// ---- DUTs/Communication/E_TaskName.TcDUT
{attribute 'qualified_only'}
{attribute 'strict'}
TYPE E_TaskName :
(
//(*
	//New
	EmptyTask :=0,
	ActivateRecipe							:=  1  	,
	ValidateRecipe                          :=  2   ,
	AlarmReset                              :=  3   ,
	ReadRFID                                :=  4   ,
	UpdateLCD                               :=  5   ,
	EnableModule                            :=  6   ,
	DisableModule                           :=  7   ,
	SetLogFileVerbosity                     :=  8   ,
	Initialize                              :=  9   ,
	Resume                                  :=  10  ,
	DoorOpen                                :=  11  ,
	DoorClose                               :=  12  ,
	DPSPower                                :=  13  ,
	UnitPresentCheck                        :=  14  ,
	TrayClamp                               :=  15  ,
	ChangeStackCount                        :=  16  ,
	BypassVision                            :=  17  ,
	TCCSessionRequest                       :=  18  ,
	TIUSlideOut                             :=  19  ,
	PrecisorSlideOut                        :=  20  ,
	SingulateTrayStacker                    :=  21  ,
	SingulateTrayStackerHalf                :=  22  ,
	SingulateTrayStackerRemaining           :=  23  ,
	StackUpTrayStacker                      :=  24  ,
	StopperUp                               :=  25  ,
	MoveConveyorForward                     :=  26  ,
	MoveConveyorBackward                    :=  27  ,
	MoveVisionShuttle                       :=  28  ,
	MoveUPortShuttle                        :=  29  ,
	UPortShuttleReady                       :=  30  ,
	MoveFlyoverShuttle                      :=  31  ,
	FlyoverShuttlePick                      :=  32  ,
	FlyoverShuttlePlace                     :=  33  ,
	MoveTrayScanShuttle                     :=  34  ,
	MoveTrayScanShuttleLifter               :=  35  ,
	EportLatch                              :=  36  ,
	GantryPickAndPlace                      :=  37  ,
	TBOTPickAndPlace                        :=  38  ,
	AutoTeach                               :=  39  ,
	Jog                                     :=  40  ,
	ApplyTeachData                          :=  41  ,
	AbortTeach                              :=  42  ,
	WriteRFIDData                           :=  43  ,
	MoveGantry                              :=  44  ,
	MoveTBOT                                :=  45  ,
	MoveTBOTRetry                           :=  46  ,
	MoveTBOTCancel                          :=  47  ,
	TBOTPickAndPlaceRetry                   :=  48  ,
	TBOTPickAndPlaceCancel                  :=  49  ,
	MoveGantryRetry                         :=  50  ,
	MoveGantryCancel                        :=  51  ,
	GantryPickAndPlaceRetry                 :=  52  ,
	GantryPickAndPlaceCancel                :=  53  ,
	SingulateTrayStackerRetry               :=  54  ,
	SingulateTrayStackerCancel              :=  55  ,
	SingulateTrayStackerHalfRetry           :=  56  ,
	SingulateTrayStackerHalfCancel          :=  57  ,
	SingulateTrayStackerRemainingRetry      :=  58  ,
	SingulateTrayStackerRemainingCancel     :=  59  ,
	StackUpTrayStackerRetry                 :=  60  ,
	StackUpTrayStackerCancel                :=  61  ,
	MoveConveyorForwardRetry                :=  62  ,
	MoveConveyorForwardCancel               :=  63  ,
	MoveConveyorBackwardRetry               :=  64  ,
	MoveConveyorBackwardCancel              :=  65  ,
	MoveVisionShuttleRetry                  :=  66  ,
	MoveVisionShuttleCancel                 :=  67  ,
	MoveUPortShuttleRetry                   :=  68  ,
	MoveUPortShuttleCancel                  :=  69  ,
	MoveFlyoverShuttleRetry                 :=  70  ,
	MoveFlyoverShuttleCancel                :=  71  ,
	MoveTrayScanShuttleRetry                :=  72  ,
	MoveTrayScanShuttleCancel               :=  73  ,
	MoveTrayScanShuttleLifterRetry          :=  74  ,
	MoveTrayScanShuttleLifterCancel         :=  75  ,
	Cancel                                  :=  76  ,
	TIUSlideOutRetry                        :=  77  ,
	TIUSlideOutCancel                       :=  78  ,
	MoveTTSShuttle                          :=  79  ,
	MoveTTSShuttleRetry                     :=  80  ,
	MoveTTSShuttleCancel                    :=  81  ,
	SingulateTrayLatchRemaining             :=  82  ,
	SingulateTrayLatchRemainingRetry        :=  83  ,
	SingulateTrayLatchRemainingCancel       :=  84  ,
	SingulateTrayLatch                      :=  85  ,
	SingulateTrayLatchRetry                 :=  86  ,
	SingulateTrayLatchCancel                :=  87  ,
	StackUpTrayLatch                        :=  88  ,
	StackUpTrayLatchRetry                   :=  89  ,
	StackUpTrayLatchCancel                  :=  90  ,
	SingulateCylinderTray                   :=  91  ,
	SingulateCylinderTrayRetry              :=  92  ,
	SingulateCylinderTrayCancel             :=  93  ,
	StackUpCylinderTray                     :=  94  ,
	StackUpCylinderTrayRetry                :=  95  ,
	StackUpCylinderTrayCancel               :=  96  ,
	SetUPortBlinkRate                       :=  97  ,
	TBotUnitPresentCheck                    :=  98  ,
	AP240ACPOWER                            :=  99  ,
	TesterAirValve                          :=  100 ,
	APAirValve                              :=  101 ,
	DrawerUp                                :=  102 ,
	SetBlinkRate							:=  103 ,
	TIUSocketCoolingAir						:=  104	,
	StackDownTrayStacker					:=	105	,
	StackDownTrayStackerRetry				:=	106	,
	StackDownTrayStackerCancel				:=	107	,
	StackDownTrayStackerRemaining			:=	108	,
	StackDownTrayStackerRemainingRetry		:=	109	,
	StackDownTrayStackerRemainingCancel		:=	110	,
	TTSShuttlePickPlace						:=	111	,
	TTSShuttlePickPlaceCancel				:=	112	,
	TTSShuttlePickPlaceRetry				:=	113	,
	HstTbotPickAndPlace						:=	114	,
	HstTbotPickAndPlaceRetry				:=	115	,
	HstTbotPickAndPlaceCancel				:=	116	,
	StackDownTrayStackerHalf				:=	117	,
	StackDownTrayStackerHalfRetry			:=	118	,
	StackDownTrayStackerHalfCancel			:=	119	,
	SetStackerBlinkRate						:=	120	,
	Ap48DCPower								:=	121	,
	BPAirValve								:=	122	,
	APPCWValve								:=	123	,
	CellLTIMValve							:=	124	,
	MainPCWValve							:=	125	,
	MainOFAValve							:=	126	,
	CmdPower								:=	127	,
	SetSolenoidValves						:=	128	,
	Secondary24VPower						:=	131

);
END_TYPE

// ---- DUTs/Communication/ST_Command.TcDUT
TYPE ST_Command :
STRUCT
	sLogName	: STRING(81);
	eTaskName	: E_TaskName;
	eModuleID	: E_ModuleID;
	iParam		: ARRAY [1..NO_OF_INT_PARAM] OF DINT;
	sParam		: ARRAY [1..NO_OF_STRING_PARAM] OF STRING;
	bParam		: ARRAY [1..NO_OF_BOOL_PARAM] OF BOOL;
	dParam		: ARRAY [1..NO_OF_LREAL_PARAM] OF LREAL;
END_STRUCT
END_TYPE

// ---- DUTs/Communication/ST_Event.TcDUT
TYPE ST_Event :
STRUCT
	sLogName	: STRING(81);
	eEventName	: E_EventName;
	eModuleID	: E_ModuleID;
	iParam		: ARRAY [1..NO_OF_INT_PARAM] OF DINT;
	sParam		: ARRAY [1..NO_OF_STRING_PARAM] OF STRING;
	bParam		: ARRAY [1..NO_OF_BOOL_PARAM] OF BOOL; 
	dParam		: ARRAY [1..NO_OF_LREAL_PARAM] OF LREAL; 
	sFailReason	: STRING(81);
END_STRUCT
END_TYPE

// ---- DUTs/Communication/ST_EventQueue.TcDUT
TYPE ST_EventQueue :
STRUCT
	Queue: ARRAY [1..255] OF ST_Event;	//255 queue buffers
	Count: UINT := 0;
END_STRUCT
END_TYPE

// ---- DUTs/Communication/ST_TACommands.TcDUT
TYPE ST_TACommands :
STRUCT
	arrTACommands : ARRAY  [1..NO_OF_CMD_BUFFER] OF ST_Command;
		
END_STRUCT
END_TYPE

// ---- DUTs/Communication/ST_TAEvents.TcDUT
TYPE ST_TAEvents :
STRUCT
	arrTAEvents : ARRAY [1..NO_OF_EVENT_BUFFER]  OF ST_Event;
	
END_STRUCT
END_TYPE

// ---- DUTs/Enum/E_BackdoorState_1.TcDUT
TYPE E_BackdoorState_1 :
(
	eDisable := 0,
	eForce_On :=1,
	eForce_Off := 2
);
END_TYPE

// ---- DUTs/Enum/E_ModuleID_1.TcDUT
TYPE E_ModuleID_1 :
(
	eNull := 0,

//Uport
	eUport1,
	eUport2,
	eUport1Stk,
	eUport2Stk,

//Uport shuttle
	eUShuttle1,
	eUShuttle2,
	eUShuttle1Cny,
	eUShuttle2Cny,
	eUShuttle1Prk,
	eUShuttle2Prk,

//LP Lane	
	eLP1,
	eLP2,
	eLP3,
	eLP4,
	eLP5,
	eLP6,
	eLP7,
	eLP8,
	
	eLP1Stk1,
	eLP2Stk1,
	eLP3Stk1,
	eLP4Stk1,
	eLP5Stk1,
	eLP6Stk1,
	eLP7Stk1,
	eLP8Stk1,

	eLP1Stk2,
	eLP2Stk2,
	eLP3Stk2,
	eLP4Stk2,
	eLP5Stk2,
	eLP6Stk2,
	eLP7Stk2,
	eLP8Stk2,
	
		eLP1Stk1Lift,
		eLP2Stk1Lift,
		eLP3Stk1Lift,
		eLP4Stk1Lift,
		eLP5Stk1Lift,
		eLP6Stk1Lift,
		eLP7Stk1Lift,
		eLP8Stk1Lift,
	
		eLP1Stk2Lift,
		eLP2Stk2Lift,
		eLP3Stk2Lift,
		eLP4Stk2Lift,
		eLP5Stk2Lift,
		eLP6Stk2Lift,
		eLP7Stk2Lift,
		eLP8Stk2Lift,

		eLP1Stk1Cny,
		eLP2Stk1Cny,
		eLP3Stk1Cny,
		eLP4Stk1Cny,
		eLP5Stk1Cny,
		eLP6Stk1Cny,
		eLP7Stk1Cny,
		eLP8Stk1Cny,
	
		eLP1Stk2Cny,
		eLP2Stk2Cny,
		eLP3Stk2Cny,
		eLP4Stk2Cny,
		eLP5Stk2Cny,
		eLP6Stk2Cny,
		eLP7Stk2Cny,
		eLP8Stk2Cny,

	eLP1Eport,
	eLP2Eport,
	eLP3Eport,
	eLP4Eport,
	eLP5Eport,
	eLP6Eport,
	eLP7Eport,
	eLP8Eport,	

		eLP1EportStk,
		eLP2EportStk,
		eLP3EportStk,
		eLP4EportStk,
		eLP5EportStk,
		eLP6EportStk,
		eLP7EportStk,
		eLP8EportStk,
	
		eLP1EportCny,
		eLP2EportCny,
		eLP3EportCny,
		eLP4EportCny,
		eLP5EportCny,
		eLP6EportCny,
		eLP7EportCny,
		eLP8EportCny,
		
		eLP1EportGrip,
		eLP2EportGrip,
		eLP3EportGrip,
		eLP4EportGrip,
		eLP5EportGrip,
		eLP6EportGrip,
		eLP7EportGrip,
		eLP8EportGrip,		
		
	eLP1Shuttle,
	eLP2Shuttle,
	eLP3Shuttle,
	eLP4Shuttle,
	eLP5Shuttle,
	eLP6Shuttle,
	eLP7Shuttle,
	eLP8Shuttle,

//TTS
	eTTS1,
	eTTS2,

	eTTS1Prk,
	eTTS2Prk,

//Vision
	eVision1,
	eVision2,
	
	eVision1Prk,
	eVision2Prk,
	
//**********************
	eUport,
	eUportStk,
	
	eUShuttle,
	eUShuttleCny,
	eUShuttlePrk,

	eLP,
	eLPStk,
	eLPStk1,
	eLPStk2,
	eLPStkCny,
	eLPStkLift,
	eLPEport,
	
	eTTS,
	eTTSPrk,
	
	eVision,
	eVisionPrk,
	
	eLPEportLatch,
	eLPEportTTS,
	
	ePNBLatch,
	ePNBSby,
	ePNB
	
	
);
END_TYPE

// ---- DUTs/Enum/E_ProcessState.TcDUT
TYPE E_ProcessState :
(
	eUNKNOWN:=0,
	eINIT,		//During Init
	//eIDLE,
	//eIDLEAL,
	//eSETGUP,
	//eREADY,
	eAWAITGCMD,	//After Done = Idle
	eLOADG,		//Processing
    //eALARM,
	ePAUSE,		//Aft Alm Rst
	//eTARESUME,
	eALPAUSED//,	//During Alm
	//eCHECKG,
	//eCOMPLETE
	
	
);
END_TYPE

// ---- DUTs/Enum/E_ProcessStep.TcDUT
TYPE E_ProcessStep :
(
	eSeqReset:=1,
	eDataInput,
	eExecuting,
	eSeqCompleted,
	eSeqError,
	eSeqCancel	
);
END_TYPE

// ---- DUTs/Enum/E_SeqSts_1.TcDUT
TYPE E_SeqSts_1 :
(
	eNull := -1,
	eInit := 0,
	ePreSanityCheck,
	eSanityCheck,
	eSanityCheck2,
	eTrayCount,

	//hw trigger
	eMotorZVelMove,	//Velosity move
	eMotorZVelMoveTeach,
	eMotorXVelMove,
	eMotorYVelMove,
	eMotorZHalt,
	eMotorXHalt,
	eMotorYHalt,
	eMotorCnyMove,
	eMotorCnyMoveSlow,
	eMotorCnyHalt,
	
// ^^^^Skip seq step till eMotorCnyHalt^^^^

	eMotorZAbsMove,	//Absolute move
	eMotorXAbsMove,
	eMotorYAbsMove,
	eMotorZRelMove,	//Relative move
	eMotorXRelMove,
	eMotorYRelMove,
	eClamp,
	eUnclamp,
	eLatch,
	eUnlatch,
	eEportLatch,
	eEportUnlatch,
	eStopperUp,
	eStopperDwn,
	eShutterOpen,
	eShutterClose,
	
	eMotorXReset,
	eMotorYReset,
	eMotorZReset,
	
	eMotorXPowerOn,
	eMotorYPowerOn,
	eMotorZPowerOn,
	
	eMotorXHome,
	eMotorYHome,
	eMotorZHome,
	
	eMotorConyReset,
	eMotorConyPowerOn,
	eMotorConyHome,
	
	eMotorZAbsMoveSbyPos,
	eMotorZAbsMoveLatchPos,
	eMotorZAbsMoveLiftPos,
	eMotorZAbsMoveTopPos,
	eMotorZAbsMoveCountSensorPos,
	eMotorZAbsMoveEportTopPos,
	eAutoTeachCalc,
		
	
	
	eCylJackUp,
	eCylJackDown,
	
	eHomeStacker,
	eHomeConveyer,
	eHomeUport,
	
	eReset,
	eExecute,
	eAlarmed,
	
	eDone :=100
	
);
END_TYPE

// ---- DUTs/E_BackdoorState.TcDUT
TYPE E_BackdoorState :
(
	eDisable := 0,
	eForce_On :=1,
	eForce_Off := 2
);
END_TYPE

// ---- DUTs/HMI/ST_BypassTII.TcDUT
TYPE ST_BypassTII :
STRUCT
	bHMITIIByPassArray:ARRAY[1..NO_OF_TII_SENSOR] OF BOOL;
END_STRUCT
END_TYPE

// ---- DUTs/ModuleState/EnableDisable/E_State.TcDUT
TYPE E_State :
(
	// Disabled
	eDisabled :=0,
	// Enabled
	eEnabled
);
END_TYPE

// ---- DUTs/ModuleState/EnableDisable/ST_LPState.TcDUT
TYPE ST_LPState :
STRUCT
	// LoadPort module state 
	//arrLPSubModule : ARRAY [1..(.NO_OF_LANES)] OF ST_TCSubModuleState;
	
	
//	EmptyStacker : ARRAY [1..(.NO_OF_STACKERS_IN_EMPTYSTK)] OF E_State := [(.NO_OF_STACKERS_IN_EMPTYSTK)(E_State.eEnabled)];
	// Vision Shuttle 
	//VisionShuttle : E_State := E_State.eEnabled;
END_STRUCT
END_TYPE

// ---- DUTs/ModuleState/EnableDisable/ST_LPTTS_State.TcDUT
TYPE ST_LPTTS_State :
STRUCT
	// LoadPort module state , 2 LPs
	arrLoadPort: ARRAY [1..(.NO_OF_LPS)] OF ST_LPState;
	// TTS moduel state
	stTTS: ST_TTS_State;
		
END_STRUCT
END_TYPE

// ---- DUTs/ModuleState/EnableDisable/ST_TCSubModuleState.TcDUT
TYPE ST_TCSubModuleState :
STRUCT
	Tester							: E_State := E_State.eEnabled;
	TCSite							: ARRAY [1..(.NO_OF_TC_SITE)] OF ST_TCSiteState;
END_STRUCT
END_TYPE

// ---- DUTs/ModuleState/EnableDisable/ST_TCSiteState.TcDUT
TYPE ST_TCSiteState :
STRUCT
	TCU						: E_State	:= E_State.eEnabled;
	TIERII					: E_State	:= E_State.eEnabled;
END_STRUCT
END_TYPE

// ---- DUTs/ModuleState/EnableDisable/ST_TTS_State.TcDUT
TYPE ST_TTS_State :
STRUCT
	// TTS moduel state
	arrTTSLane: ARRAY [1..3] OF E_State := [(3)(E_State.eEnabled)];
END_STRUCT
END_TYPE

// ---- DUTs/ModuleState/EPT/E_EPT.TcDUT
TYPE E_EPT :
(
	// Unknown, Alarm, Paused, Aborting, Claibration, Manual
	eBlocked :=0,
	// Idle
	eIdle,
	// Initialize, SettingUp, Ready, Executing, Checking
	eBusy 
);
END_TYPE

// ---- DUTs/ModuleState/EPT/ST_LPTTS_EPT.TcDUT
TYPE ST_LPTTS_EPT :
STRUCT
	// LoadPort module state , 2 LPs
	//arrLoadPort: ARRAY [1..(.NO_OF_LPS)] OF ST_LP_EPT;
	// TTS moduel state
	stTTS: ST_TTS_EPT;
		
END_STRUCT
END_TYPE

// ---- DUTs/ModuleState/EPT/ST_TCUEPT.TcDUT
TYPE ST_TCUEPT :
STRUCT
	// LoadPort module state 
	//arrLPSubModule : ARRAY [1..(.NO_OF_LANES)] OF ST_LP_SubModuleEPT;
	// Vision Shuttle 
	TCU : E_EPT;
END_STRUCT
END_TYPE

// ---- DUTs/ModuleState/EPT/ST_TCSubModuleEPT.TcDUT
TYPE ST_TCSubModuleEPT :
STRUCT
	TCSite: ARRAY [1..(.NO_OF_TC_SITE)] OF ST_TCUEPT;
END_STRUCT
END_TYPE

// ---- DUTs/ModuleState/EPT/ST_TC_EPT.TcDUT
TYPE ST_TC_EPT :
STRUCT
	eTCEpt:E_EPT;
	
END_STRUCT
END_TYPE

// ---- DUTs/ModuleState/EPT/ST_TTS_EPT.TcDUT
TYPE ST_TTS_EPT :
STRUCT
	// TTS State
	eTTS: E_EPT;
	// TTS moduel state
	arrTTSLane: ARRAY [1..3] OF E_EPT;
END_STRUCT
END_TYPE

// ---- DUTs/ST_StepMode.TcDUT
TYPE ST_StepMode :
STRUCT
	bStepMode: BOOL;  //module in step mode
	bStep	 : BOOL;  //Step by step
END_STRUCT
END_TYPE

// ---- DUTs/ST_DebugStation.TcDUT
TYPE ST_DebugStation :
STRUCT
		stGblDBStnParam		: ST_DebugStationSeqParam;
		fbDBStnSeq			: FB_DebugStationSeq;
END_STRUCT
END_TYPE

// ---- DUTs/ST_TCMultilevel.TcDUT
TYPE ST_TCMultilevel :
STRUCT
	
		stGblParam							: ST_TCMultiLevelSeqParam;
		fbTCMultiLevelSeq					: FB_TCMultiLevelSeq;
		
END_STRUCT
END_TYPE

// ---- DUTs/ST_TCShuttlePOC.TcDUT
TYPE ST_TCShuttlePOC :
STRUCT
	
		stGblParam: ST_TCSeqParam;
		fbTCShuttlePOCSeq: FB_TCShuttlePOCSeq;

END_STRUCT
END_TYPE

// ---- DUTs/ST_TCLevel.TcDUT
TYPE ST_TCLevel :
STRUCT
	
		stGblParam: ST_TCSeqParam;
		fbTCLevelSeq: FB_TCLevelSeq;
		
END_STRUCT
END_TYPE

// ---- GVLs/GVL_CONSTANTS.TcGVL
VAR_GLOBAL CONSTANT

	// This function has been automatically generated from the project information.
	stLibVersion_TC : ST_LibVersion := (iMajor := 0, iMinor := 0, iBuild := 0, iRevision := 0, sVersion := '2.0.5');

	LA_LEVEL_MODULE_ID : ARRAY [1..NO_OF_LEVEL] OF E_ModuleID  := [	E_ModuleID.CELL_LA101_TESTER, E_ModuleID.CELL_LA201_TESTER, E_ModuleID.CELL_LA301_TESTER,
																	E_ModuleID.CELL_LA401_TESTER, E_ModuleID.CELL_LA501_TESTER, E_ModuleID.CELL_LA601_TESTER];
	LB_LEVEL_MODULE_ID : ARRAY [1..NO_OF_LEVEL] OF E_ModuleID  := [	E_ModuleID.CELL_LB101_TESTER, E_ModuleID.CELL_LB201_TESTER, E_ModuleID.CELL_LB301_TESTER,
																	E_ModuleID.CELL_LB401_TESTER, E_ModuleID.CELL_LB501_TESTER, E_ModuleID.CELL_LB601_TESTER];
	LC_LEVEL_MODULE_ID : ARRAY [1..NO_OF_LEVEL] OF E_ModuleID  := [	E_ModuleID.CELL_LC101_TESTER, E_ModuleID.CELL_LC201_TESTER, E_ModuleID.CELL_LC301_TESTER,
																	E_ModuleID.CELL_LC401_TESTER, E_ModuleID.CELL_LC501_TESTER, E_ModuleID.CELL_LC601_TESTER];
	RA_LEVEL_MODULE_ID : ARRAY [1..NO_OF_LEVEL] OF E_ModuleID  := [	E_ModuleID.CELL_RA101_TESTER, E_ModuleID.CELL_RA201_TESTER, E_ModuleID.CELL_RA301_TESTER,
																	E_ModuleID.CELL_RA401_TESTER, E_ModuleID.CELL_RA501_TESTER, E_ModuleID.CELL_RA601_TESTER];
	RB_LEVEL_MODULE_ID : ARRAY [1..NO_OF_LEVEL] OF E_ModuleID  := [	E_ModuleID.CELL_RB101_TESTER, E_ModuleID.CELL_RB201_TESTER, E_ModuleID.CELL_RB301_TESTER,
																	E_ModuleID.CELL_RB401_TESTER, E_ModuleID.CELL_RB501_TESTER, E_ModuleID.CELL_RB601_TESTER];
	RC_LEVEL_MODULE_ID : ARRAY [1..NO_OF_LEVEL] OF E_ModuleID  := [	E_ModuleID.CELL_RC101_TESTER, E_ModuleID.CELL_RC201_TESTER, E_ModuleID.CELL_RC301_TESTER,
																	E_ModuleID.CELL_RC401_TESTER, E_ModuleID.CELL_RC501_TESTER, E_ModuleID.CELL_RC601_TESTER];	
														
	LA_FRONT_DOOR_MODULE_ID : ARRAY [1..2] OF E_ModuleID  := [E_ModuleID.CELL_LA101_TESTER_FRONT, E_ModuleID.CELL_LA201_TESTER_FRONT];	
	
//<ForEnDisMod>
	ARR_LA_TST_MODULE_ID : ARRAY [1..6] OF E_ModuleID  := [E_ModuleID.CELL_LA101_TESTER, E_ModuleID.CELL_LA201_TESTER, E_ModuleID.CELL_LA201_TESTER, 
														   E_ModuleID.CELL_LA401_TESTER, E_ModuleID.CELL_LA501_TESTER, E_ModuleID.CELL_LA601_TESTER];	
	ARR_LB_TST_MODULE_ID : ARRAY [1..6] OF E_ModuleID  := [E_ModuleID.CELL_LB101_TESTER, E_ModuleID.CELL_LB201_TESTER, E_ModuleID.CELL_LB201_TESTER, 
														   E_ModuleID.CELL_LB401_TESTER, E_ModuleID.CELL_LB501_TESTER, E_ModuleID.CELL_LB601_TESTER];	
	ARR_LC_TST_MODULE_ID : ARRAY [1..6] OF E_ModuleID  := [E_ModuleID.CELL_LC101_TESTER, E_ModuleID.CELL_LC201_TESTER, E_ModuleID.CELL_LC201_TESTER, 
														   E_ModuleID.CELL_LC401_TESTER, E_ModuleID.CELL_LC501_TESTER, E_ModuleID.CELL_LC601_TESTER];															   
	ARR_RA_TST_MODULE_ID : ARRAY [1..6] OF E_ModuleID  := [E_ModuleID.CELL_RA101_TESTER, E_ModuleID.CELL_RA201_TESTER, E_ModuleID.CELL_RA201_TESTER, 
													   	   E_ModuleID.CELL_RA401_TESTER, E_ModuleID.CELL_RA501_TESTER, E_ModuleID.CELL_RA601_TESTER];	
	ARR_RB_TST_MODULE_ID : ARRAY [1..6] OF E_ModuleID  := [E_ModuleID.CELL_RB101_TESTER, E_ModuleID.CELL_RB201_TESTER, E_ModuleID.CELL_RB201_TESTER, 
													       E_ModuleID.CELL_RB401_TESTER, E_ModuleID.CELL_RB501_TESTER, E_ModuleID.CELL_RB601_TESTER];	
	ARR_RC_TST_MODULE_ID : ARRAY [1..6] OF E_ModuleID  := [E_ModuleID.CELL_RC101_TESTER, E_ModuleID.CELL_RC201_TESTER, E_ModuleID.CELL_RC201_TESTER, 
														   E_ModuleID.CELL_RC401_TESTER, E_ModuleID.CELL_RC501_TESTER, E_ModuleID.CELL_RC601_TESTER];		
														   
	ARR_LA_TCU_MODULE_ID : ARRAY [1..6] OF E_ModuleID  := [E_ModuleID.CELL_LA101_AP, E_ModuleID.CELL_LA201_AP, E_ModuleID.CELL_LA201_AP, 
														   E_ModuleID.CELL_LA401_AP, E_ModuleID.CELL_LA501_AP, E_ModuleID.CELL_LA601_AP];	
	ARR_LB_TCU_MODULE_ID : ARRAY [1..6] OF E_ModuleID  := [E_ModuleID.CELL_LB101_AP, E_ModuleID.CELL_LB201_AP, E_ModuleID.CELL_LB201_AP, 
														   E_ModuleID.CELL_LB401_AP, E_ModuleID.CELL_LB501_AP, E_ModuleID.CELL_LB601_AP];	
	ARR_LC_TCU_MODULE_ID : ARRAY [1..6] OF E_ModuleID  := [E_ModuleID.CELL_LC101_AP, E_ModuleID.CELL_LC201_AP, E_ModuleID.CELL_LC201_AP, 
														   E_ModuleID.CELL_LC401_AP, E_ModuleID.CELL_LC501_AP, E_ModuleID.CELL_LC601_AP];															   
	ARR_RA_TCU_MODULE_ID : ARRAY [1..6] OF E_ModuleID  := [E_ModuleID.CELL_RA101_AP, E_ModuleID.CELL_RA201_AP, E_ModuleID.CELL_RA201_AP, 
													   	   E_ModuleID.CELL_RA401_AP, E_ModuleID.CELL_RA501_AP, E_ModuleID.CELL_RA601_AP];	
	ARR_RB_TCU_MODULE_ID : ARRAY [1..6] OF E_ModuleID  := [E_ModuleID.CELL_RB101_AP, E_ModuleID.CELL_RB201_AP, E_ModuleID.CELL_RB201_AP, 
													       E_ModuleID.CELL_RB401_AP, E_ModuleID.CELL_RB501_AP, E_ModuleID.CELL_RB601_AP];	
	ARR_RC_TCU_MODULE_ID : ARRAY [1..6] OF E_ModuleID  := [E_ModuleID.CELL_RC101_AP, E_ModuleID.CELL_RC201_AP, E_ModuleID.CELL_RC201_AP, 
														   E_ModuleID.CELL_RC401_AP, E_ModuleID.CELL_RC501_AP, E_ModuleID.CELL_RC601_AP];		


	ARR_LA_TII_MODULE_ID : ARRAY [1..6] OF E_ModuleID  := [E_ModuleID.CELL_LA101_TIERII, E_ModuleID.CELL_LA201_TIERII, E_ModuleID.CELL_LA201_TIERII, 
														   E_ModuleID.CELL_LA401_TIERII, E_ModuleID.CELL_LA501_TIERII, E_ModuleID.CELL_LA601_TIERII];	
	ARR_LB_TII_MODULE_ID : ARRAY [1..6] OF E_ModuleID  := [E_ModuleID.CELL_LB101_TIERII, E_ModuleID.CELL_LB201_TIERII, E_ModuleID.CELL_LB201_TIERII, 
														   E_ModuleID.CELL_LB401_TIERII, E_ModuleID.CELL_LB501_TIERII, E_ModuleID.CELL_LB601_TIERII];	
	ARR_LC_TII_MODULE_ID : ARRAY [1..6] OF E_ModuleID  := [E_ModuleID.CELL_LC101_TIERII, E_ModuleID.CELL_LC201_TIERII, E_ModuleID.CELL_LC201_TIERII, 
														   E_ModuleID.CELL_LC401_TIERII, E_ModuleID.CELL_LC501_TIERII, E_ModuleID.CELL_LC601_TIERII];															   
	ARR_RA_TII_MODULE_ID : ARRAY [1..6] OF E_ModuleID  := [E_ModuleID.CELL_RA101_TIERII, E_ModuleID.CELL_RA201_TIERII, E_ModuleID.CELL_RA201_TIERII, 
													   	   E_ModuleID.CELL_RA401_TIERII, E_ModuleID.CELL_RA501_TIERII, E_ModuleID.CELL_RA601_TIERII];	
	ARR_RB_TII_MODULE_ID : ARRAY [1..6] OF E_ModuleID  := [E_ModuleID.CELL_RB101_TIERII, E_ModuleID.CELL_RB201_TIERII, E_ModuleID.CELL_RB201_TIERII, 
													       E_ModuleID.CELL_RB401_TIERII, E_ModuleID.CELL_RB501_TIERII, E_ModuleID.CELL_RB601_TIERII];	
	ARR_RC_TII_MODULE_ID : ARRAY [1..6] OF E_ModuleID  := [E_ModuleID.CELL_RC101_TIERII, E_ModuleID.CELL_RC201_TIERII, E_ModuleID.CELL_RC201_TIERII, 
														   E_ModuleID.CELL_RC401_TIERII, E_ModuleID.CELL_RC501_TIERII, E_ModuleID.CELL_RC601_TIERII];		
														   
//</ForEnDisMod>														  


													
	ARR_AMS_NET_ID : ARRAY [1..NO_OF_COLUMN] OF STRING := [	'192.168.1.4.1.1',
															'192.168.1.5.1.1', 
															'192.168.1.6.1.1',
															'192.168.1.14.1.1',
															'192.168.1.15.1.1', 
															'192.168.1.16.1.1'];	
		
	ARR_COL_MOD_ID : ARRAY [1..NO_OF_COLUMN] OF E_ModuleID := [	E_ModuleID.COLUMN_LA,
																E_ModuleID.COLUMN_LB,
																E_ModuleID.COLUMN_LC,
																E_ModuleID.COLUMN_RA,
																E_ModuleID.COLUMN_RB,
																E_ModuleID.COLUMN_RC];										
	TIIAlmText : ARRAY[1..NO_OF_TII_SENSOR] OF STRING :=
	[
	 	'AP_Not_Present'					,	
	 	'APPower_Not_On'	    			,
	 	'AP_Not_Ready' 		    			,
	 	'APDeactuatedPLC_Not_On' 			,
	 	'APDeactuatedHwr_Not_On' 			,
	 	'CellFluid_Leakage1' 				,
	 	'CellFluid_Leakage2' 				,
	 	'Cell_GroundFault' 					,
	 	'Tester_Not_Present' 				,
	 	'TesterPower_Not_On' 				,
	 	'Tester_not_ready'					,
	 	'TCCellDoor_Not_Locked'				,
	 	'TesterLatches_Not_Closed' 			,
	 	'TBOT_TC_ACPower_Off_Signal' 		,
		'DS_Facility_EAP_ACPower_Signal'	,
		'FrontDoorLockSignalNotDetected'	,
	 	'TCDrawerCylExtendRS_Not_On' 		,
	 	'TCDrawerCylRetractRS_Not_On'		,
		'TCDrawerUpSignal_not_on'			,
		'TCDrawerDownSignal_not_on'		    	
	];
	
	EAPAlmText : ARRAY[1..NO_OF_LEVEL,1..NO_OF_EAP_ALARM] OF STRING :=
	[
	 	'TBOT EAP ALARM_1'				,	
	 	'TBOT EAP ALARM_2'				,
	 	'TBOT EAP ALARM_3'				,
	 	'TBOT EAP ALARM_4'				,
	 	'TBOT EAP ALARM_5'				,
	 	'TBOT EAP ALARM_6'				,
	 	'TBOT EAP ALARM_7'				,
	 	'TBOT EAP ALARM_8'				,
	 	'TBOT EAP ALARM_9'				,
	 	'TBOT EAP ALARM_10'			
	];
	 
	SysAlmText : ARRAY[1..NO_OF_COMMON_SENSOR] OF STRING :=
	[
	 	'Column_PCWLeakage',
	 	'AllTCDrawer_Not_In_Cell',       
	 	'ipTbotDoorClosedSignal'
	];
	
	DBStnSysAlmText : ARRAY[1..NO_OF_DBCOL_ALARM] OF STRING :=
	[
	 	'SystemPCWLeakageAlarm',
	 	'SystemPCWSupplyLeakageAlarm',       
	 	'SystemPCWReturnLeakageAlarm',
	 	'CriticalCondensationAlarm',
	 	'6BarLowOFAAirPressureAlarm'
	];
															
	NO_OF_COMMON_SENSOR 						: UINT	:= 3;
	NO_OF_TII_SENSOR 							: UINT	:= 30;
	NO_OF_ALARM_TAG								: UINT 	:= 50;
	NO_OF_DC_CELL_LEVEL							: UINT	:= 2;
	NO_OF_LEVEL 								: UINT 	:= 6;
	NO_OF_COLUMN 								: UINT 	:= 6;
	NO_OF_TC_SITE								: UINT	:= 1;
	NO_OF_SENSORS 								: UINT 	:= 20;
	NO_OF_BTNLED								: INT	:= 5;
	NO_OF_EAP_ALARM								: INT	:= 10;
	NO_OF_DBCOL_ALARM							: INT	:= 10;
	
	//Path Setting
	LOGFILEPATHTC1 :STRING(30) := 'D:/ControllerLog/Level1/';
	LOGFILEPATHTC2 :STRING(30) := 'D:/ControllerLog/Level2/';
	LOGFILEPATHTC3 :STRING(30) := 'D:/ControllerLog/Level3/';
	LOGFILEPATHTC4 :STRING(30) := 'D:/ControllerLog/Level4/';
	LOGFILEPATHTC5 :STRING(30) := 'D:/ControllerLog/Level5/';
	
	//Log verbosity
	LOG_LEVEL_ERROR   : INT := 5;
	LOG_LEVEL_WARNING : INT := 4;
	LOG_LEVEL_MESSAGE : INT := 3;
	LOG_LEVEL_INFO    : INT := 2;
	LOG_LEVEL_DEBUG   : INT := 1;
	
	NO_OF_CMD_BUFFER : INT := 30;
	NO_OF_EVENT_BUFFER : INT := 30;
		
	NO_OF_INT_PARAM : INT := 10;
	NO_OF_STRING_PARAM :INT := 5;
	NO_OF_BOOL_PARAM :INT := 32;
	NO_OF_LREAL_PARAM :INT := 10;


	MODULEID_ERROR : STRING := 'Module ID not correct';

	NO_OF_LIB_ALARM:INT:=30;
	NO_OF_TA_ALARM: INT:=100;
	NO_OF_ALARM_PER_LEVEL : INT := 100;
END_VAR
VAR_GLOBAL
	lrTest: REAL;
END_VAR

// ---- GVLs/GVL_EAP.TcGVL
//{attribute 'qualified_only'}
VAR_GLOBAL
	stEAP:ST_EAP;
	stDCEAP:ST_DCEAP;
	DS_Facility_eapShutOffAllACPower					AT %I* :BOOL; // shut off Tester and AP AC Power, 0: On, 1: Off //only for debug cart and station
END_VAR

// ---- GVLs/GVL_Motor.TcGVL
//{attribute 'qualified_only'}
VAR_GLOBAL
	GVL_DUT_TC_AP240ACPower					: DUT_Cylinder;
	GVL_DUT_DC_AP240ACPower					: DUT_Cylinder;
END_VAR

// ---- GVLs/GVL_Process.TcGVL
//{attribute 'qualified_only'}
VAR_GLOBAL
	Sec_P						: BOOL;
	DewPoint_Warning			: BOOL;
	DewPoint_Alarm				: BOOL;
	DewPoint_Abort				: BOOL;
	OFA6Bar_Warning				: BOOL;
	OFA6Bar_Alarm				: BOOL;
	OFA6Bar_Abort				: BOOL;
	
	DewPoint_Warning_Timer		: UDINT	:= 300;
	DewPoint_Alarm_Timer		: UDINT	:= 60;
	DewPoint_Abort_Timer		: UDINT	:= 60;
	OFA6Bar_Warning_Timer		: UDINT	:= 300;
	OFA6Bar_Alarm_Timer			: UDINT	:= 60;
	OFA6Bar_Abort_Timer			: UDINT	:= 60;
	
	DewPoint_LowSP				: LREAL	:= 2;
	DewPoint_LowLowSP			: LREAL	:= 0;
	OFA6Bar_LowSP				: LREAL	:= 550;
	OFA6Bar_LowLowSP			: LREAL	:= 500;
END_VAR

// ---- GVLs/GVL_SEN_SPEC.TcGVL
//{attribute 'qualified_only'}
VAR_GLOBAL
	
sen1Spec :ST_SenSpec := (iMn :=0, iMx :=0, oMn :=0, oMx :=0, ofs :=0, b:=0);

//	65535 			->  32768  	-> 	16384.
//	a/5 = 13107 	-> 	6553.5 	-> 	3276.75
// *0.6 = 7864.2 	->  3932.1  ->  1966.05

spDBStnTstAirLeakFlowSensor 		:ST_SenSpec := (iMn :=0, 	iMx :=32768, oMn :=0 	 , oMx :=0.1 , ofs :=0		, b:=0.0); //0  - 	10V	|	0     - 0.1 l/min
spDBStnAPAirLeakFlowSensor			:ST_SenSpec := (iMn :=0, 	iMx :=32768, oMn :=0 	 , oMx :=0.1 , ofs :=0		, b:=0.0); //0 	- 	10V	|	0     - 0.1 l/min
spDBStnPCWLeakFlowSensor 			:ST_SenSpec := (iMn :=0, 	iMx :=32768, oMn :=0	 , oMx :=65	 , ofs :=0		, b:=0.0); //0 	- 	10V	|	0     - 65 	ml/min (Rabiah)
spDBStnPCWLowFlowSensor 			:ST_SenSpec := (iMn :=3276, iMx :=16384, oMn :=0	 , oMx :=4	 , ofs :=0		, b:=0.0); //1 	- 	5V	| 	0     - 4  	l/min
                                                                                         
spDBColumnPCWRegularFlowSensor		:ST_SenSpec := (iMn :=3276, iMx :=16384, oMn :=0	 , oMx :=100 , ofs :=0		, b:=0.0); //1	-	5V	|	0     - 100 l/min
spDBColumnPCWSupplyPressure       	:ST_SenSpec := (iMn :=3276, iMx :=16384, oMn :=0	 , oMx :=10	 , ofs :=0		, b:=0.0); //1	-	5V	|	0     - 1 MPa
spDBColumnPCWReturnPressure       	:ST_SenSpec := (iMn :=3276, iMx :=16384, oMn :=0	 , oMx :=10	 , ofs :=0		, b:=0.0); //1	-	5V	|	0  	  - 1 MPa
spDBColumnTstAirPressure          	:ST_SenSpec := (iMn :=1966, iMx :=16384, oMn :=-1	 , oMx :=10	 , ofs :=0		, b:=0.0); //0.6-	5V	|	-0.1  - 1MPa     1MPa = 10 bar
spDBColumnAPAirPressure           	:ST_SenSpec := (iMn :=1966, iMx :=16384, oMn :=-1	 , oMx :=10	 , ofs :=0		, b:=0.0); //0.6-	5V	|	-0.1  - 1MPa
spDBColumnDewPointSensor          	:ST_SenSpec := (iMn :=3276, iMx :=16384, oMn :=-40	 , oMx :=60	 , ofs :=0		, b:=0.0); //1	-	5V	|	-40   - 60 ˚C
spDBColumnTempSensor	          	:ST_SenSpec := (iMn :=3276, iMx :=16384, oMn :=-40	 , oMx :=60	 , ofs :=0		, b:=0.0); //1	-	5V	|	-40   - 60 ˚C

// Thermocouple
spDBColumnPCWSupplyTemperature    	:ST_SenSpec := (iMn :=-400, iMx :=2500, oMn :=-40, oMx :=250, ofs :=0, b:=0.0); //	Ask Spec
spDBColumnPCWReturnTemperature    	:ST_SenSpec := (iMn :=-400, iMx :=2500, oMn :=-40, oMx :=250, ofs :=0, b:=0.0); //

//EL3314 Spec
//Temperature range in the range defined in each case for the sensor (default setting: type K; -200…+1370 °C); voltage measurement: ±30 mV…±75 mV
//Resolution:	0.1 °C per digit
//Conversion time:	approx. 2.5 s up to 20 ms, depending on configuration and filter setting, default: approx. 250 ms

lmtPCWSupplyHighTempWarning_Limit 			:REAL := 14 ;	//14
lmt6BarLowOFAAirPressureWarning_Limit 		:REAL := 550 ;	//550
lmt9BarLowOFAAirPressureWarning_limit 		:REAL := 850 ;	//850
lmtExcessiveHeatLoadIntoPCWWarning_Limit 	:REAL := 14 ;	//14
lmtCondensationWarning_Limit				:REAL := -2 ;	//-2
lmtCriticalCondensationAlarm_Limit			:REAL := 0 ;	//0

END_VAR

// ---- GVLs/GVL_TA.TcGVL
VAR_GLOBAL
	// 1 = Production mode, 0 = Engineering mode 
	// Engineering mode can have IO's from either of one, Actual HW , Backdoor or Simualted
	bProductionMode										: BOOL	:= TRUE;  //0: simulation, 1: actual/ production mode
	bEnableTIIAlarm										: BOOL	:= FALSE;
	
	// TA Heartbeat signal 
	bTAHeartBeat										: BOOL; (* ~ (OPC : 1 : available for OPC-Clients) 
										  						(OPC_PROP[0005] : 3 : OPC_PROP_RIGHTS, here Read Write*)
								
	// PLC Heartbeat signal 
	bTCSHeartBeat										: BOOL; 		
	// False: aTCS reading in progress , clear array  and toggle to true once done. TA stop sending commands
	// True: TCS Ready to receive cmd data. TA: Sending commands and toggle to false once done
	arrTCSCommandReady									: BOOL; //arrTCSReady
	iTCSReady											: INT; 	//-	IntAlignmentWithTBotPNB 1/Nov/18	
	
	// Receive commands from TA 
	arrTACommands										: ST_TACommands ;
	// False: TCS updating events and toggelr to true once done, TA stop reading events  
	// True: TCS stop updating events, TA start copy events and clear, toggle to false once done.
	arrTCSEventTriggered								: BOOL;
	iTCSEventTriggered									: INT;	//-	IntAlignmentWithTBotPNB 1/Nov/18	
							
	// Event send back from TCS to TA
	arrTCSEvents:  ST_TAEvents;
																	
	bDiagnosticMode 									: BOOL;
	bColIODiagnosticsMode								: BOOL;
	arrIODiagnosticsMode								: ARRAY [1..(.NO_OF_LEVEL)] OF BOOL	:= [(.NO_OF_LEVEL)(FALSE)];
	
	// TC: Enable /Disable State
	//arrTCLevelState: ARRAY [1..(.NO_OF_LEVEL)] OF E_State :=[(NO_OF_LEVEL)(E_State.eEnabled)];
	TC_ModuleState										: ARRAY[1..NO_OF_LEVEL] OF ST_TCSubModuleState;
	
	// TC: EPT States(Blocked, idle, busy)
	//arrTCMLevelEpt:ARRAY[1..NO_OF_LEVEL] OF E_EPT;	
	TC_EPT 												: ARRAY [1..NO_OF_LEVEL] OF ST_TCSubModuleEPT;
	//ALMTC: ST_AlarmSubmodules;
	ALMTC												: ST_AlarmModules;
	
//<DC COLUMN>
	ALM_DBSTN											: ST_AlarmTags;
	ALM_DCCOL											: ST_AlarmTags;
//</DC COLUMN>
	
	arrStepMode											: ARRAY[1..NO_OF_LEVEL] OF ST_StepMode;
	
	bMainAirValve										: BOOL	:= TRUE;
END_VAR

// ---- GVLs/GVL_TC.TcGVL
VAR_GLOBAL
	COLUMN_NAME 							: E_ModuleID	:= E_ModuleID.COLUMN_LC;
	bGetAMSNetID							: BOOL;
	IsNetIDReadOK							: BOOL	:= FALSE;
	LevelModuleID							: ARRAY [1..NO_OF_LEVEL] OF E_ModuleID;
	
//<Optional Flag>
	bDebugStation							: BOOL := FALSE; // T : Do Debug Station Action
	bDebugCart								: BOOL := TRUE;	// T : Do Debug Cart Action
	bAnalogIOSim 							: BOOL := FALSE;
	bAlwaysOnAPPwrOnInit  					: BOOL; // F : if(!present)skip pwrOnStep, T : Doesn't depends on present signal. 
	bAlwaysOnTstPwrOn 						: BOOL;
	bSLTC									: BOOL; // T : SLTC
	bEnableManualCommandTest1 				: BOOL := FALSE; // Manual Command Test from PLC level (recommanded only for trained person)
	bEnableManualCommandTest2 				: BOOL := FALSE;
//</Optional Flag>
	
//<DefaultValueContainer>	
	BtnSetTstPwrOnChkDelay 					: BOOL	:= FALSE;
	BtnSetAPPwrOnChkDelay 					: BOOL	:= FALSE;
	iTstPwrOnChkDelay						: INT	:= 0;
	iAPPwrOnChkDelay						: INT	:= 0;
	TstPwrOnChkDelay						: TIME	:= T#20S;
	APPwrOnChkDelay							: TIME	:= T#1S;
	TstPrstChkDelay							: TIME	:= T#1S;
	APPrstChkDelay							: TIME	:= T#1S;
	DispTstPwrOnChkDelay					: INT;
	DispAPPwrOnChkDelay						: INT;
	
	BtnSetTstReadyCheckDelay 				: BOOL	:= FALSE;
	BtnSetAPReadyCheckDelay 				: BOOL	:= FALSE;
	iTstReadyCheckDelay						: INT	:= 0;
	iAPReadyCheckDelay						: INT	:= 0;
	TstReadyCheckDelay						: TIME	:= T#20S;
	APReadyCheckDelay						: TIME	:= T#1S;
	DispTstReadyCheckDelay					: INT;
	DispAPReadyCheckDelay					: INT;
	
	
	tDwrCylExtRetSensorDelay				: TIME	:= T#200MS;
	tDwrCylUpDownSensorDelay				: TIME	:= T#200MS;
	tDwrCylExtRetTimeOut					: TIME	:= T#7000MS;
	tDwrCylUpDownTimeOut					: TIME	:= T#4000MS;
//<DefaultValueContainer>

	iTCColumnID								: UINT:=1;
	//iPOC_ML_Selection:INT:=2; 	//1:POC: 2:Multilevel
	//IsTIIAlarms  :ARRAY[1..NO_OF_LEVEL] OF BOOL;
	//IsSysAlarm : BOOL;

	arrTCShuttlePOC 						: ARRAY [1..NO_OF_LEVEL] OF ST_TCShuttlePOC;
	arrTCVIO 								: ARRAY [1..2] OF ST_TCShuttlePOC_VIO;
	
	arrTCLevel 								: ARRAY [1..1] OF ST_TCLevel; //for SLTC only
	arrTCLevelVIO 							: ARRAY [1..NO_OF_LEVEL] OF ST_TCLevel_VIO;
	//arrDPSPower: ARRAY [1..NO_OF_LEVEL] OF BOOL; //for SLTC only
	
	arrTCMultiLevel 						: ARRAY [1..NO_OF_LEVEL] OF ST_TCMultilevel; //for MLTC only
	arrTCMultiLevelVIO 						: ARRAY [1..NO_OF_LEVEL] OF ST_TCMultiLevel_VIO;
	
	stGblDbStnVIO 							: ST_DebugStation_VIO;
	
	//TIIAlmText : ARRAY[1..NO_OF_TII_SENSOR] OF STRING;
	//SysAlmText : ARRAY[1..NO_OF_COMMON_SENSOR] OF STRING;
	
	stDebugStation 							: ST_DebugStation;//FB_DebugStation
	fbDebugColumn  							: FB_DebugColumn;
	fbDbStnTIIAlarm 						: FB_TIIAlarmDbStn;
	
	//ModuleType : E_TCModuleType //ALPHA_TC,DEBUG_CART,SLTC,SLTC_POC,SLTC_CX16,
	//EnableColumnSensorCheck for //SLTC TC(s) and DebugCarts
	//EnableSideDoors //for DebugCarts
	//En/Dis Some TII for SLTC(s)
	//En/Dis Some TII for DC
	
	fbTCColumn								: FB_TCColumn; //for MLTC only
	arrTIIAlarm 							: ARRAY [1..NO_OF_LEVEL] OF FB_TIIAlarm;
	
	fbSLTCExtra 							: FB_SLTC_EXTA;
	
	
	iLogVerbosity 							: INT	:= LOG_LEVEL_DEBUG;
	
	
	//REMOTE COMMAND and Events
	// Receive commands from TA  are just copied in this array and then from here further divided
	// based on level
	arrCommands								: (*ARRAY [1..(.NO_OF_LEVEL)] OF*) ST_TACommands;
	//Empty structure of command
	stEmptyCommand							: ST_Command;
	// Event send back to TA are just copied in this array and then from here further divided
	// based on level
	
	
	//ArrAlarmCode: ARRAY [1..4] OF ST_AlarmFault;
	//
	arrEvents								: (*ARRAY [1..(.NO_OF_LEVEL)] OF*) ST_TAEvents;
	// To store alarm and other asynchronous events that require busy state
	arrPendingEventsQueue					: (*ARRAY [1..(.NO_OF_LEVEL)] OF*) ST_EventQueue;
	//Empty event structure
	stEmptyEvents							: ST_Event;
	
	//Once TCS recieves Connect command this turns true: else false
	//When true TCS starts follwoing heart beat signal from TA
	bTAConnected							: BOOL	:= FALSE;
	bAlarmEnabled							: BOOL	:= FALSE;

	// If event updation ongoing
	arrEventUpdating						: BOOL;
	
	aiXConverted							: ARRAY [1..NO_OF_LEVEL] OF REAL;
	aiYConverted							: ARRAY [1..NO_OF_LEVEL] OF REAL;
	aiY1Converted							: ARRAY [1..NO_OF_LEVEL] OF REAL;
	aiZConverted							: ARRAY [1..NO_OF_LEVEL] OF REAL;

	aiXConvertedRet							: ARRAY [1..NO_OF_LEVEL] OF REAL;
	aiYConvertedRet							: ARRAY [1..NO_OF_LEVEL] OF REAL;
	aiZConvertedRet							: ARRAY [1..NO_OF_LEVEL] OF REAL;
	
	bMoveShuttle							: BOOL;	
	fbFormat								: FB_FormatString;

	//ArrAlmBitBefDelay : ARRAY[1..200] OF BOOL;
	//ArrAlmBitAftDelay : ARRAY[1..200] OF BOOL;
	//ArrAlarmKeepBit	:	ARRAY[1..200] OF BOOL;
	//ArrDelayAlarm : 	ARRAY[1..200] OF FB_DelayAlarm;
	//Arr_ms :			ARRAY[1..200] OF INT;
	
	
//<HMI_Control>
	bHMIRsetEvntTriggerOnProductionMode		: BOOL;
	iHMIBtnType:int;
	arrHMIBtnSolidOn_Condition				: ARRAY[1..NO_OF_LEVEL, 0..NO_OF_BTNLED - 1] OF BOOL;
	

	
	bHMIBtnSimulation						: BOOL;	// Must be False on Actual RUN; For manual Button Simulation
	stHMIBtnSimArray						: ARRAY [1..NO_OF_LEVEL] OF ST_BypassTII;
	
	bHMIEnTIISenSimulation					: BOOL;// Must be False on Actual RUN; System Alm Sen and TII Alm Sen
	stHMITIISenSimArray						: ARRAY [1..NO_OF_LEVEL] OF ST_BypassTII;
	bHMIColSenSimArray						: ARRAY [1..NO_OF_COMMON_SENSOR] OF BOOL;
	
	bHMITIIBypass							: BOOL	:= FALSE; // HMI TII Bypass Check Box.
	stHMITIIByPassArray						: ARRAY[1..NO_OF_LEVEL] OF ST_BypassTII;
	arrHMISysAlmByPass						: ARRAY[1..NO_OF_COMMON_SENSOR] OF BOOL;
	
	bHMIResetAllAlarm						: BOOL	:= FALSE;
	iHMICbLevelSelection					: INT	:= 1;
	iHMICbCmdSelection						: INT	:= 1;
//</HMI_Control>
	FunONOFF								: BOOL;
	
	bSimulation								: BOOL;
	GetRand									: dRAND;
END_VAR

// ---- POUs/3) FB/2) TC/Testing/CycleTest.TcPOU
PROGRAM CycleTest
VAR
	bCycleStart1:BOOL:= FALSE;
	bCycleStart2:BOOL:= FALSE;
	LevelToStart:INT:=3;
	iLevel:INT:=1;
	iNoOfLevel:INT:=4; //NO_OF_LEVEL;
	nState:INT;
	nCount:INT:=1;
	fbGUI_TEST : ARRAY [1..NO_OF_LEVEL] OF FB_GUI_TEST;
	arrLevelStartBits :ARRAY[1..NO_OF_LEVEL] OF BOOL;
	
	TDelay : TON;
	TDelay1: TON;
	TDelay2 : TON;
	ClearTCSEvent: TON;
	tCaptureDelay: TIME:= T#1000MS;
	tDelayNextStep: TIME:= T#2000MS;
	tInterval: TIME:= T#200MS;
	tempstr :STRING;
	i:INT;
	iClearCount: INT;
	iTotalClear: INT:=20;
	
	nNoOfCyclePerLevel:INT:=1;
	bStartCycle	:BOOL;
	bStart		:BOOL;
	stVIO :ST_TCMultiLevel_VIO;
	isError:BOOL;
	
	arrCount:ARRAY[1..NO_OF_LEVEL] OF INT;
	NoOfCycCount:INT :=5;
END_VAR

//<region>
	CASE nState OF
		0:
			nState:=1;
			iLevel:=LevelToStart;
		1:
			IF bCycleStart1 AND bCycleStart2 THEN 
				nState:=2; 
			ELSE
				IF bCycleStart1 XOR bCycleStart2 THEN
					bCycleStart1:=FALSE;
					bCycleStart2:=FALSE;
				END_IF
				iLevel:=LevelToStart;
			END_IF
		2:
			arrLevelStartBits[iLevel]:=TRUE;
			nState:=3;
		3:	stVIO:=arrTCMultiLevel[iLevel].fbTCMultiLevelSeq.stMLVIO;
			
			IF bCycleStart1 AND bCycleStart2 AND NOT isError THEN
				arrTCSEventTriggered :=FALSE;
				fbGUI_TEST[iLevel](iLevel:=iLevel,nCount:=nCount,bStart:=arrLevelStartBits[iLevel]);
				isError:= stVIO.isTIIError OR stVIO.isSysError OR arrTCMultiLevel[iLevel].fbTCMultiLevelSeq.P_bError;
				IF NOT arrLevelStartBits[iLevel] THEN 
					arrCount[iLevel]:=arrCount[iLevel]+1;
					Logging.fbDebugLog.M_nLogger(1, sSource:='LEVEL CYCLE COUNT', F_concat3('Level',F_concat3('[',INT_TO_STRING(iLevel), ']'), F_concat3('Cycle Count =',', ',INT_TO_STRING(arrCount[iLevel]) ) ) );
					IF iLevel < iNoOfLevel THEN
						iLevel:=iLevel+1;
						nState:=4;
					ELSIF iLevel >= iNoOfLevel THEN
						IF arrCount[iLevel]>=NoOfCycCount THEN
							arrCount[iLevel]:=0;
							bCycleStart1:=bCycleStart2 := FALSE;
						END_IF
						iLevel:=LevelToStart;
						nState:=4;
					END_IF
				END_IF	
			END_IF
			IF isError THEN
				isError:= stVIO.isTIIError OR stVIO.isSysError OR arrTCMultiLevel[iLevel].fbTCMultiLevelSeq.P_bError;
			END_IF
		4:
			nState:=1;
		5:	
		
	END_CASE
	

//</region>

(*
//<CycleTest02>
	CASE nState OF
		0:
			TDelay(IN:=FALSE);
	 		TDelay1(IN:=FALSE);
			TDelay2(IN:=FALSE);
			i:=1;
			nState:=1;
		1:
			IF bCycleStart1 AND bCycleStart2 THEN 
				nState:=2; 
			ELSE
				IF bCycleStart1 XOR bCycleStart2 THEN
					bCycleStart1:=FALSE;
					bCycleStart2:=FALSE;
				END_IF
				iLevel:=1;
			END_IF
		2:
			arrLevelStartBits[iLevel]:=TRUE;
			nState:=3;
		3:
			arrTACommands.arrTACommands[1].sLogName := CONCAT('TIUSlideOut_TESTER_LA':CONCAT('0':INT_TO_STRING(iLevel)));
			arrTACommands.arrTACommands[1].eTaskName := E_TaskName.TIUSlideOut;
			arrTACommands.arrTACommands[1].eModuleID := LEVEL_MODULE_ID[iLevel];
			arrTACommands.arrTACommands[1].bParam[1] := TRUE;
			arrTCSCommandReady:= FALSE;
			iClearCount := iTotalClear;
			
			ClearTCSEvent(IN:=(iClearCount > 0): PT:=T#100MS);
			IF ClearTCSEvent.Q THEN
				ClearTCSEvent(IN:=FALSE);
				iClearCount := iClearCount - 1;
				arrTCSEventTriggered:= FALSE;
			END_IF
			nState:=4;
		4:	
			IF arrTCMultiLevel[iLevel].stGblParam.bShuttleMoveOut =FALSE THEN
				TDelay1(IN:=TRUE:PT:=tCaptureDelay);
				IF TDelay1.Q THEN
					TDelay2(IN:=TRUE:PT:=tInterval);
					IF TDelay2.Q THEN
											
						TDelay2(IN:=FALSE);
						tempstr[1] := F_concat3('X: ': REAL_TO_STRING(aiXConverted): ': ');
						tempstr[2] := F_concat3('Y: ': REAL_TO_STRING(aiYConverted): ': ');
						tempstr[3] := F_concat3('Z: ': REAL_TO_STRING(aiZConverted): ': ');
						
						tempstr[4] := F_concat3(tempstr[1]: tempstr[2]: tempstr[3]);
						Logging.fbDebugLog.M_nLogger(1: sSource:='aisensor': F_concat3(INT_TO_STRING(i): ': ': tempstr[4]));
						i := i+1;
					END_IF
				END_IF
				TDelay(IN:=TRUE:PT:=tDelayNextStep);//after move out: delay before move in
				IF TDelay.Q THEN
					TDelay(IN:=FALSE);
					nState := 2;
				END_IF
			END_IF
		5:	//Move In
			arrTACommands.arrTACommands[1].sLogName := CONCAT('TIUSlideOut_TESTER_LA':CONCAT('0':INT_TO_STRING(iLevel)));
			arrTACommands.arrTACommands[1].eTaskName := E_TaskName.TIUSlideOut;
			arrTACommands.arrTACommands[1].eModuleID := LEVEL_MODULE_ID[iLevel];
			arrTACommands.arrTACommands[1].bParam[1] := TRUE;
			arrTCSCommandReady:= FALSE;
			iClearCount := iTotalClear;
			
			ClearTCSEvent(IN:=(iClearCount > 0): PT:=T#100MS);
			IF ClearTCSEvent.Q THEN
				ClearTCSEvent(IN:=FALSE);
				iClearCount := iClearCount - 1;
				arrTCSEventTriggered:= FALSE;
			END_IF
			nState:=4;
			nState := 6;
		6:	//
			IF arrTCMultiLevel[iLevel].stGblParam.bShuttleMoveIn=FALSE THEN
		    	TDelay(IN:=TRUE:PT:=tDelayNextStep);//after move out: delay before move in
		    	IF TDelay.Q THEN
		    		TDelay(IN:=FALSE);
		    		nState := 0;
		    		nCount := nCount +1;
		    	END_IF	 
		    END_IF
		7:  
				IF nCount> nNoOfCyclePerLevel(*AND nState =3*) THEN
		arrLevelStartBits[iLevel] := FALSE;
		bStart:=FALSE;
		nCount:=1;
		//bPBStart := FALSE;
		
	END_IF
		
		8:	
			
			IF NOT arrLevelStartBits[iLevel] THEN 
				IF iLevel < NO_OF_LEVEL THEN
					iLevel:=iLevel+1;
					nState:=4;
				ELSIF iLevel >= NO_OF_LEVEL THEN
					iLevel:=1;
					nState:=4;
				END_IF
			END_IF	
		9:
			nState:=0;
		
	END_CASE
//</CycleTest02>
*)

END_PROGRAM

// ---- POUs/3) FB/2) TC/Testing/FB_GUI_TEST.TcPOU
FUNCTION_BLOCK FB_GUI_TEST
VAR_INPUT
	iLevel :INT;
	nCount: INT:=0;
END_VAR
VAR
	bInitialise : BOOL := FALSE;
	bStartCycle : BOOL := FALSE;
	tCaptureDelay: TIME:= T#1000MS;
	tDelayNextStep: TIME:= T#200MS;
	tInterval: TIME:= T#250MS;
	
	bCylinderUp : BOOL;
	//iLevel : UINT :=2; 
	
	nState : UINT :=0;
	//nCount: INT:=0;
	nNoOfCycle:INT:=1;
	TDelay : TON;
	TDelay1 : TON;
	bUp: BOOL;
	sErr: STRING;
	tempstr : ARRAY[1..4] OF STRING;
	tempstrRet : ARRAY[1..4] OF STRING;
	str: STRING;
	TDelay2 : TON;
	i: INT :=1;
	
	bCylinderOutL1: BOOL;
	bOutL1 : BOOL;
	
	bPBStart : BOOL;
	
	StartPbDly: TON;
	rtStartTrig :R_Trig;
	
	
	iClearCount: INT;
	iTotalClear: INT:=20;
	ClearTCSEvent: TON;
	mlVIO:ST_TCMultiLevel_VIO; 
END_VAR
VAR_IN_OUT
	bStart:BOOL;
END_VAR

IF bInitialise THEN
	arrTCMultiLevel[iLevel].stGblParam.bInitialise:=TRUE;
	bInitialise:=FALSE;
END_IF

IF bCylinderUp THEN
	IF (arrTCMultiLevel[iLevel].fbTCMultiLevelSeq.M_nCmptUpDown(bUp, sErr)=10) THEN
		bCylinderUp :=FALSE;
	END_IF
END_IF

IF bCylinderOutL1 THEN
	IF (arrTCMultiLevel[iLevel].fbTCMultiLevelSeq.M_nCmptInOut(bOutL1, sErr)=10) THEN
		bCylinderOutL1 :=FALSE;
	END_IF
END_IF

(*StartPbDly(in:=(stIO[iLevel].ipStartPB),pt:=T#100MS);
rtStartTrig(Clk:=StartPbDly.Q);
IF rtStartTrig.Q THEN
	bPBStart:=TRUE;
END_IF *)

bPBStart := arrTCVIO[iLevel].ipStartPB;

IF bStartCycle XOR bStart THEN //cycle Up down, in out
	CASE nState OF
		0: //Out
	 		TDelay(IN:=FALSE);
	 		TDelay1(IN:=FALSE);
			TDelay2(IN:=FALSE);
			i:=1;
			nState := 1;
		1: //Out
	 		//TDelay(IN:=FALSE);
	 		//TDelay1(IN:=FALSE);
			//TDelay2(IN:=FALSE);
			//i:=1;
			//arrTCMultiLevel[iLevel].stGblParam.bShuttleMoveOut := TRUE;
			//<MoveOut>
				arrTACommands.arrTACommands[1].sLogName := CONCAT('TIUSlideOut_TESTER_LA',CONCAT('0',INT_TO_STRING(iLevel)));
				arrTACommands.arrTACommands[1].eTaskName := E_TaskName.TIUSlideOut;
				arrTACommands.arrTACommands[1].eModuleID := LevelModuleID[iLevel];
				arrTACommands.arrTACommands[1].bParam[1] := TRUE;
				arrTCSCommandReady:= FALSE;
				iClearCount := iTotalClear;
				
				ClearTCSEvent(IN:=(iClearCount > 0), PT:=T#100MS);
				IF ClearTCSEvent.Q THEN
					ClearTCSEvent(IN:=FALSE);
					iClearCount := iClearCount - 1;
					arrTCSEventTriggered:= FALSE;
				END_IF
			//</region>
			
	 		nState := 2;
	 2:		mlVIO:= arrTCMultiLevel[iLevel].fbTCMultiLevelSeq.P_stTCMultiLevelVIO;
			IF mlVIO.ipTCDrawerCylExtendRS= TRUE THEN
	 			nState := 3;
			END_IF
	 //Delay					
	 3: 	IF arrTCMultiLevel[iLevel].stGblParam.bShuttleMoveOut =FALSE THEN
		    	IF iLevel = 3 THEN   // Level No for Distance Laser Sensor Reading
		 			TDelay1(IN:=TRUE,PT:=tCaptureDelay);
					IF TDelay1.Q THEN
						TDelay2(IN:=TRUE,PT:=tInterval);
						IF TDelay2.Q THEN			
							TDelay2(IN:=FALSE);
							tempstr[1] := F_concat3('XE,', REAL_TO_STRING(aiXConverted[iLevel]), ', ');
							tempstr[2] := F_concat3('YE,', REAL_TO_STRING(aiYConverted[iLevel]), ', ');
							tempstr[3] := F_concat3('ZE,', REAL_TO_STRING(aiZConverted[iLevel]), ', ');
							tempstr[4] := F_concat3(tempstr[1], tempstr[2], tempstr[3]);
							
							tempstrRet[1] := F_concat3('XR,', REAL_TO_STRING(aiXConvertedRet[iLevel]), ', ');
							tempstrRet[2] := F_concat3('YR,', REAL_TO_STRING(aiYConvertedRet[iLevel]), ', ');
							tempstrRet[3] := F_concat3('ZR,', REAL_TO_STRING(aiZConvertedRet[iLevel]), ', ');
							tempstrRet[4] := F_concat3(tempstrRet[1], tempstrRet[2], tempstrRet[3]);
							
							str:= '';
							str:= CONCAT(tempstr[4] , tempstrRet[4]);
							Logging.fbDebugLog.M_nLogger(1, sSource:='aisensor', F_concat3(INT_TO_STRING(i), ', ', str));
							
							//Logging.fbDebugLog.M_nLogger(1, sSource:='aisensor', F_concat3(INT_TO_STRING(i), ', ', tempstr[4]));
							i := i+1;
							IF i>4 THEN
								nState := 4;
							END_IF
						END_IF
						//END_FOR
					END_IF
					(*
					TDelay(IN:=TRUE,PT:=tDelayNextStep);//after move out, delay before move in
					IF TDelay.Q THEN
						TDelay(IN:=FALSE);
						nState := 3;
					END_IF
					*)
					
				ELSE
					nState := 4;
				END_IF
				
			END_IF

	 4:		//In
			//arrTCMultiLevel[iLevel].stGblParam.bShuttleMoveIn := TRUE;
	 		//<MoveIn>
				arrTACommands.arrTACommands[1].sLogName := CONCAT('TIUSlideOut_TESTER_LA',CONCAT('0',INT_TO_STRING(iLevel)));
				arrTACommands.arrTACommands[1].eTaskName := E_TaskName.TIUSlideOut;
				arrTACommands.arrTACommands[1].eModuleID := LevelModuleID[iLevel];
				arrTACommands.arrTACommands[1].bParam[1] := FALSE;
				arrTCSCommandReady:= FALSE;
				iClearCount := iTotalClear;
				
				ClearTCSEvent(IN:=(iClearCount > 0), PT:=T#100MS);
				IF ClearTCSEvent.Q THEN
					ClearTCSEvent(IN:=FALSE);
					iClearCount := iClearCount - 1;
					arrTCSEventTriggered:= FALSE;
				END_IF
			//</MoveIn>
			
	 		nState := 5;
			
	5:
	 		mlVIO:= arrTCMultiLevel[iLevel].fbTCMultiLevelSeq.P_stTCMultiLevelVIO;
			IF mlVIO.ipTCDrawerCylRetractRS= TRUE THEN
	 			nState := 6;
			END_IF
			//Done
	 6: 	IF arrTCMultiLevel[iLevel].stGblParam.bShuttleMoveIn=FALSE THEN
			TDelay(IN:=TRUE,PT:=tDelayNextStep);//after move out, delay before move in
			IF TDelay.Q THEN
				TDelay(IN:=FALSE);
				nState := 0;
				nCount := nCount +1;
			END_IF	 
	 
			END_IF
	END_CASE
	
	IF nCount> nNoOfCycle(*AND nState =3*) THEN
		bStartCycle := FALSE;
		bStart:=FALSE;
		nCount:=1;
		//bPBStart := FALSE;
		
	END_IF
		
END_IF

END_FUNCTION_BLOCK

// ---- DUTs/Logging/F_Concat5.TcPOU
FUNCTION F_Concat5 : STRING(255)
VAR_INPUT
	sString1: STRING(255);
	sString2: STRING(255);
	sString3: STRING(255);
	sString4: STRING(255);
	sString5: STRING(255);
END_VAR

F_Concat5 := CONCAT(F_Concat5, sString1);
F_Concat5 := CONCAT(F_Concat5, sString2);
F_Concat5 := CONCAT(F_Concat5, sString3);
F_Concat5 := CONCAT(F_Concat5, sString4);
F_Concat5 := CONCAT(F_Concat5, sString5);

END_FUNCTION

// ---- POUs/2) DFB/Facility/DFB_FacilityAlarmAnlg.TcPOU
FUNCTION_BLOCK DFB_FacilityAlarmAnlg
VAR_INPUT
	Sec_P					: BOOL; // Second pulse
	PV						: LREAL; // Process Value
	WarningTimer			: UDINT;
	AlarmTimer				: UDINT;
	AbortTimer				: UDINT;
	DB						: LREAL	:= 0.2; // Deadband
	LogName					: STRING;
	ModuleID				: E_ModuleID;
	EventName				: E_EventName;
	E_FacilityState			: E_FacilityState;
END_VAR

VAR_OUTPUT
	Warning					: BOOL;
	Alarm					: BOOL;
	Abort					: BOOL;
END_VAR

VAR_IN_OUT
	LowSP					: LREAL; // Low Alarm Set Point
	LowLowSP				: LREAL; // Low Low Alarm Set Point
END_VAR

VAR
	_State_Changed			: BOOL;
	
	_State					: INT;
	_Last_State				: INT;
	_TLast_State			: INT;
	
	_AbortStateTimer			: UDINT;
	_WarningStateTimer		: UDINT;
	_AlarmStateTimer		: UDINT;
	_WarningActive			: BOOL;
	_AlarmActive			: BOOL;
	_AbortActive			: BOOL;
	
	_EmptyEvent				: ST_Event;
END_VAR

///////////////////////////////////////////////////////////////////////////////////////////////////////////////////////////////////////////////////////////////////////////////
//	State timer
///////////////////////////////////////////////////////////////////////////////////////////////////////////////////////////////////////////////////////////////////////////////

_State_Changed									:= _State <> _TLast_State;
_TLast_State									:= _State;

IF _State_Changed THEN
	Logging.fbDebugLog.M_nLogger(iLogLevel:= iLogVerbosity, sSource:= 'AIN Log', 
		sMessage								:= CONCAT(CONCAT(LogName, 'current state['),
														 CONCAT(INT_TO_STRING(_State), ']'))); 
END_IF

IF Sec_P THEN
	IF _WarningActive AND _WarningStateTimer < WarningTimer THEN
		_WarningStateTimer					:= _WarningStateTimer+1;
	END_IF
	
	IF _AlarmActive AND _AlarmStateTimer < AlarmTimer THEN
		_AlarmStateTimer					:= _AlarmStateTimer+1;
	END_IF
	
	IF _AbortActive AND _AbortStateTimer < AbortTimer THEN
		_AbortStateTimer					:= _AbortStateTimer+1;
	END_IF
END_IF


IF NOT _WarningActive THEN
	_WarningStateTimer						:= 0;
END_IF
IF NOT _AlarmActive THEN
	_AlarmStateTimer						:= 0;
END_IF

IF NOT _AbortActive THEN
	_AbortStateTimer						:= 0;
END_IF


///////////////////////////////////////////////////////////////////////////////////////////////////////////////////////////////////////////////////////////////////////////////
//	Safety clamp
///////////////////////////////////////////////////////////////////////////////////////////////////////////////////////////////////////////////////////////////////////////////

IF LowSP < LowLowSP THEN
	LowSP										:= LowLowSP;
END_IF

///////////////////////////////////////////////////////////////////////////////////////////////////////////////////////////////////////////////////////////////////////////////
//	State case
///////////////////////////////////////////////////////////////////////////////////////////////////////////////////////////////////////////////////////////////////////////////

CASE _State OF
	0: (*Idle*)
	
		(*Action*)
		Warning									:= FALSE;
		Alarm									:= FALSE;
		Abort									:= FALSE;
		
		_AlarmActive							:= FALSE;
		_WarningActive							:= FALSE;
		_AbortActive							:= FALSE;
		
		(*Transition*)
		IF PV < LowLowSP THEN
			_State								:= 21; // Low Low Alarm - Delay
			_AlarmActive						:= TRUE;
			_WarningActive						:= TRUE;
		ELSIF PV < LowSP THEN
			_State								:= 11; // Low Alarm - Delay
			_WarningActive						:= TRUE;
		END_IF
		
	11: (*Low Alarm - Delay*)
		_Last_State								:= 11;
		
		(*Action*)
		Warning									:= TRUE;
		Alarm									:= FALSE;
		Abort									:= FALSE;
		
		(*Transition*)
		IF PV >= LowSP + DB THEN
			_State								:= 0; // Idle
		ELSIF PV < LowLowSP THEN
			_State								:= 21; // Low Low Alarm - Delay
			_AlarmActive						:= TRUE;
		ELSIF _WarningStateTimer >= WarningTimer THEN
			_State								:= 22; // Low Alarm - Send Event
		END_IF
	
	21: (*Low Low Alarm - Delay*)
		_Last_State								:= 21;
		
		(*Action*)
		Warning									:= TRUE;
		Alarm									:= TRUE;
		Abort									:= FALSE;
		
		(*Transition*)
		IF PV >= LowLowSP + DB THEN
			_State								:= 0; // Idle
		ELSIF _AlarmStateTimer >= AlarmTimer THEN
			_State								:= 24; // Low Low Alarm - Send Event
		ELSIF _WarningStateTimer >= WarningTimer THEN
			_State								:= 24; // Low Alarm - Send Event (to prevent warning timer is shorter than Alarm timer when both alarm and warning are active)
		END_IF
	
	22:	(*Low Alarm - Send Event*)
		_Last_State								:= 22;
		
		(*Action*)
		Warning									:= TRUE;
		Alarm									:= FALSE;
		Abort									:= FALSE;
		
		// Event - AbortInProgress
		CmdAndEventProcess.fbCmdAndEventUpdate.M_AddEvent(
			sLogName							:= LogName, 
			eEventName							:= EventName, 
			eModuleID							:= ModuleID, 
			iParam								:= _EmptyEvent.iParam,
			sParam								:= _EmptyEvent.sParam, 
			bParam								:= _EmptyEvent.bParam, 
			dParam								:= _EmptyEvent.dParam,
			sFailReason							:= '');
		
		(*Transition*)
		_State									:= 25; // Low Low Alarm - Check abort time
		_AbortActive							:= TRUE;
		
	24: (*Low Low Alarm - Send Event*)
		_Last_State								:= 24;
		
		(*Action*)
		Warning									:= TRUE;
		Alarm									:= TRUE;
		Abort									:= FALSE;
		
		// Event - AbortInProgress
		CmdAndEventProcess.fbCmdAndEventUpdate.M_AddEvent(
			sLogName							:= LogName, 
			eEventName							:= EventName, 
			eModuleID							:= ModuleID, 
			iParam								:= _EmptyEvent.iParam,
			sParam								:= _EmptyEvent.sParam, 
			bParam								:= _EmptyEvent.bParam, 
			dParam								:= _EmptyEvent.dParam,
			sFailReason							:= '');
		
		(*Transition*)
		_State									:= 26; // Low Low Alarm - Check abort time
		_AbortActive							:= TRUE;
		
	25: (*Low Alarm - Abort Delay*)
		_Last_State								:= 25;
		
		(*Action*)
		Warning									:= TRUE;
		Alarm									:= FALSE;
		Abort									:= FALSE;
		
		(*Transition*)
		IF _AbortStateTimer >= AbortTimer THEN
			_State								:= 40; // Abort
		END_IF
		
	26: (*Low Low Alarm - Abort Delay*)
		_Last_State								:= 26;
		
		(*Action*)
		Warning									:= TRUE;
		Alarm									:= TRUE;
		Abort									:= FALSE;
		
		(*Transition*)
		IF _AbortStateTimer >= AbortTimer THEN
			_State								:= 41; // Abort
		END_IF
		
	40: (*Low Alarm - Abort*)
		_Last_State								:= 40;
		
		(*Action*)
		Warning									:= TRUE;
		Alarm									:= FALSE;
		Abort									:= TRUE;
		
		(*Transition*)
		IF PV >= LowSP + DB THEN
			_State								:= 0; // Idle
		END_IF
		
	41: (*Lowlow Alarm - Abort*)
		_Last_State								:= 41;
		
		(*Action*)
		Warning									:= TRUE;
		Alarm									:= TRUE;
		Abort									:= TRUE;
		
		(*Transition*)
		IF PV >= LowSP + DB THEN
			_State								:= 0; // Idle
		END_IF
END_CASE

END_FUNCTION_BLOCK

// ---- POUs/2) DFB/Facility/DFB_FacilityAlarm.TcPOU
FUNCTION_BLOCK DFB_FacilityAlarm
VAR_INPUT
	Sec_P					: BOOL; // Second pulse
	PV						: LREAL; // Process Value
	WarningTimer			: UDINT;
	AlarmTimer				: UDINT;
	AbortTimer				: UDINT;
	DB						: LREAL	:= 0.2; // Deadband
	LogName					: STRING;
	ModuleID				: E_ModuleID;
	EventName				: E_EventName;
END_VAR

VAR_OUTPUT
	Warning					: BOOL;
	Alarm					: BOOL;
	Abort					: BOOL;
END_VAR

VAR_IN_OUT
	LowSP					: LREAL; // Low Alarm Set Point
	LowLowSP				: LREAL; // Low Low Alarm Set Point
END_VAR

VAR
	_State_Changed			: BOOL;
	
	_State					: INT;
	_Last_State				: INT;
	_TLast_State			: INT;
	
	_State_Timer			: UDINT;
	
	
	_EmptyEvent				: ST_Event;
END_VAR

///////////////////////////////////////////////////////////////////////////////////////////////////////////////////////////////////////////////////////////////////////////////
//	State timer
///////////////////////////////////////////////////////////////////////////////////////////////////////////////////////////////////////////////////////////////////////////////

_State_Changed									:= _State <> _TLast_State;
_TLast_State									:= _State;

IF _State_Changed THEN
	_State_Timer								:= 0;
	Logging.fbDebugLog.M_nLogger(iLogLevel:= iLogVerbosity, sSource:= 'AIN Log', 
		sMessage								:= CONCAT(CONCAT(LogName, 'current state['),
														 CONCAT(INT_TO_STRING(_State), ']'))); 
	
ELSE
	IF Sec_P THEN
		_State_Timer							:= _State_Timer + 1;
	END_IF
END_IF


///////////////////////////////////////////////////////////////////////////////////////////////////////////////////////////////////////////////////////////////////////////////
//	Safety clamp
///////////////////////////////////////////////////////////////////////////////////////////////////////////////////////////////////////////////////////////////////////////////

IF LowSP < LowLowSP THEN
	LowSP										:= LowLowSP;
END_IF

///////////////////////////////////////////////////////////////////////////////////////////////////////////////////////////////////////////////////////////////////////////////
//	State case
///////////////////////////////////////////////////////////////////////////////////////////////////////////////////////////////////////////////////////////////////////////////

CASE _State OF
	0: (*Idle*)
	
		(*Action*)
		Warning									:= FALSE;
		Alarm									:= FALSE;
		Abort									:= FALSE;
		
		(*Transition*)
		IF PV < LowLowSP THEN
			_State								:= 21; // Low Low Alarm - Delay
		ELSIF PV < LowSP THEN
			_State								:= 11; // Low Alarm - Delay
		END_IF
		
	11: (*Low Alarm - Delay*)
		_Last_State								:= 11;
		
		(*Action*)
		Warning									:= TRUE;
		Alarm									:= FALSE;
		Abort									:= FALSE;
		
		(*Transition*)
		IF PV >= LowSP + DB THEN
			_State								:= 0; // Idle
		ELSIF PV < LowLowSP THEN
			_State								:= 21; // Low Low Alarm - Delay
		ELSIF _State_Timer >= WarningTimer THEN
			_State								:= 22; // Low Low Alarm - Delay
		END_IF
	
	21: (*Low Low Alarm - Delay*)
		_Last_State								:= 21;
		
		(*Action*)
		Warning									:= TRUE;
		Alarm									:= TRUE;
		Abort									:= FALSE;
		
		(*Transition*)
		IF PV >= LowSP + DB THEN
			_State								:= 0; // Idle
		ELSIF _State_Timer >= AlarmTimer THEN
			_State								:= 24; // Low Low Alarm - Send Event
		END_IF
	
	22:	(*Low Alarm - Send Event*)
		_Last_State								:= 22;
		
		(*Action*)
		Warning									:= TRUE;
		Alarm									:= FALSE;
		Abort									:= FALSE;
		
		// Event - AbortInProgress
		CmdAndEventProcess.fbCmdAndEventUpdate.M_AddEvent(
			sLogName							:= LogName, 
			eEventName							:= EventName, 
			eModuleID							:= ModuleID, 
			iParam								:= _EmptyEvent.iParam,
			sParam								:= _EmptyEvent.sParam, 
			bParam								:= _EmptyEvent.bParam, 
			dParam								:= _EmptyEvent.dParam,
			sFailReason							:= '');
		
		(*Transition*)
		_State									:= 25; // Low Low Alarm - Check abort time
		
	24: (*Low Low Alarm - Send Event*)
		_Last_State								:= 24;
		
		(*Action*)
		Warning									:= TRUE;
		Alarm									:= TRUE;
		Abort									:= FALSE;
		
		// Event - AbortInProgress
		CmdAndEventProcess.fbCmdAndEventUpdate.M_AddEvent(
			sLogName							:= LogName, 
			eEventName							:= EventName, 
			eModuleID							:= ModuleID, 
			iParam								:= _EmptyEvent.iParam,
			sParam								:= _EmptyEvent.sParam, 
			bParam								:= _EmptyEvent.bParam, 
			dParam								:= _EmptyEvent.dParam,
			sFailReason							:= '');
		
		(*Transition*)
		_State									:= 26; // Low Low Alarm - Check abort time
		
	25: (*Low Alarm - Check abort time*)
		_Last_State								:= 25;
		
		(*Action*)
		Warning									:= TRUE;
		Alarm									:= FALSE;
		Abort									:= FALSE;
		
		(*Transition*)
		IF _State_Timer >= AbortTimer THEN
			_State								:= 40; // Abort
		END_IF
		
	26: (*Low Low Alarm - Check abort time*)
		_Last_State								:= 26;
		
		(*Action*)
		Warning									:= TRUE;
		Alarm									:= TRUE;
		Abort									:= FALSE;
		
		(*Transition*)
		IF _State_Timer >= AbortTimer THEN
			_State								:= 41; // Abort
		END_IF
		
	40: (*Abort*)
		_Last_State								:= 40;
		
		(*Action*)
		Warning									:= TRUE;
		Alarm									:= FALSE;
		Abort									:= TRUE;
		
		(*Transition*)
		IF PV >= LowSP + DB THEN
			_State								:= 0; // Idle
		END_IF
		
	41: (*Abort*)
		_Last_State								:= 41;
		
		(*Action*)
		Warning									:= TRUE;
		Alarm									:= TRUE;
		Abort									:= TRUE;
		
		(*Transition*)
		IF PV >= LowSP + DB THEN
			_State								:= 0; // Idle
		END_IF
END_CASE

END_FUNCTION_BLOCK

// ---- POUs/2) DFB/Facility/DFB_FacilityAlarm_1.TcPOU
FUNCTION_BLOCK DFB_FacilityAlarm_1
VAR_INPUT
	Sec_P					: BOOL; // Second pulse
	TbotNo					: INT; // 1: Tbot left, 2: Tbot right
	PV						: LREAL; // Process Value
	WarningTimer			: UDINT;
	AlarmTimer				: UDINT;
	AbortTimer				: UDINT;
	DB						: LREAL	:= 0.2; // Deadband
	LogName					: STRING;
	ModuleID				: E_ModuleID;
	EventName				: E_EventName;
END_VAR

VAR_OUTPUT
	Warning					: BOOL;
	Alarm					: BOOL;
	Abort					: BOOL;
END_VAR

VAR_IN_OUT
	LowSP					: LREAL; // Low Alarm Set Point
	LowLowSP				: LREAL; // Low Low Alarm Set Point
END_VAR

VAR
	_State_Changed			: BOOL;
	
	_State					: INT;
	_Last_State				: INT;
	_TLast_State			: INT;
	
	_State_Timer			: UDINT;
	
	
	_EmptyEvent				: ST_Event;
	
	_TON_Warning			: TON;
	_TON_Alarm				: TON;		
END_VAR

///////////////////////////////////////////////////////////////////////////////////////////////////////////////////////////////////////////////////////////////////////////////
//	State timer
///////////////////////////////////////////////////////////////////////////////////////////////////////////////////////////////////////////////////////////////////////////////

_State_Changed									:= _State <> _TLast_State;
_TLast_State									:= _State;

IF _State_Changed THEN
	_State_Timer								:= 0;
	Logging.fbDebugLog.M_nLogger(iLogLevel:= iLogVerbosity, sSource:= 'AIN Log', 
		sMessage								:= CONCAT(CONCAT(LogName, 'current state['),
														 CONCAT(INT_TO_STRING(_State), ']'))); 
	
ELSE
	IF Sec_P THEN
		_State_Timer							:= _State_Timer + 1;
	END_IF
END_IF


///////////////////////////////////////////////////////////////////////////////////////////////////////////////////////////////////////////////////////////////////////////////
//	Safety clamp
///////////////////////////////////////////////////////////////////////////////////////////////////////////////////////////////////////////////////////////////////////////////

IF LowSP < LowLowSP THEN
	LowSP										:= LowLowSP;
END_IF

///////////////////////////////////////////////////////////////////////////////////////////////////////////////////////////////////////////////////////////////////////////////
//	State case
///////////////////////////////////////////////////////////////////////////////////////////////////////////////////////////////////////////////////////////////////////////////

CASE _State OF
	0: (*Idle*)
	
		(*Action*)
		Warning									:= FALSE;
		Alarm									:= FALSE;
		Abort									:= FALSE;
		_TON_Warning(IN:= FALSE, PT:= UDINT_TO_TIME(WarningTimer * 1000));
		
		(*Transition*)
		IF PV < LowLowSP THEN
			_TON_Warning(IN:= TRUE, PT:= UDINT_TO_TIME(WarningTimer * 1000));
			_State								:= 21; // Low Low Alarm - Delay
		ELSIF PV < LowSP THEN
			_TON_Warning(IN:= TRUE, PT:= UDINT_TO_TIME(WarningTimer * 1000));
			_State								:= 11; // Low Alarm - Delay
		END_IF
		
	11: (*Low Alarm - Delay*)
		_Last_State								:= 11;
		
		(*Action*)
		Warning									:= TRUE;
		Alarm									:= FALSE;
		Abort									:= FALSE;
		
		(*Transition*)
		IF PV >= LowSP + DB THEN
			_State								:= 0; // Idle
		ELSIF PV < LowLowSP THEN
			_State								:= 21; // Low Low Alarm - Delay
		ELSIF _State_Timer >= WarningTimer THEN
			_State								:= 22; // Low Alarm - Send Event
		END_IF
	
	21: (*Low Low Alarm - Delay*)
		_Last_State								:= 21;
		
		(*Action*)
		Warning									:= FALSE;
		Alarm									:= TRUE;
		Abort									:= FALSE;
		
		(*Transition*)
		IF PV >= LowSP + DB THEN
			_State								:= 0; // Idle
		ELSIF _State_Timer >= AlarmTimer THEN
			_State								:= 24; // Low Low Alarm - Send Event
		END_IF
	
	22:	(*Low Alarm - Send Event*)
		_Last_State								:= 22;
		
		(*Action*)
		Warning									:= TRUE;
		Alarm									:= FALSE;
		Abort									:= FALSE;
		
		// Event - AbortInProgress
		CmdAndEventProcess.fbCmdAndEventUpdate.M_AddEvent(
			sLogName							:= LogName, 
			eEventName							:= EventName, 
			eModuleID							:= ModuleID, 
			iParam								:= _EmptyEvent.iParam,
			sParam								:= _EmptyEvent.sParam, 
			bParam								:= _EmptyEvent.bParam, 
			dParam								:= _EmptyEvent.dParam,
			sFailReason							:= '');
		
		(*Transition*)
		_State									:= 25; // Low Alarm - Check abort time
		
	24: (*Low Low Alarm - Send Event*)
		_Last_State								:= 24;
		
		(*Action*)
		Warning									:= FALSE;
		Alarm									:= TRUE;
		Abort									:= FALSE;
		
		// Event - AbortInProgress
		CmdAndEventProcess.fbCmdAndEventUpdate.M_AddEvent(
			sLogName							:= LogName, 
			eEventName							:= EventName, 
			eModuleID							:= ModuleID, 
			iParam								:= _EmptyEvent.iParam,
			sParam								:= _EmptyEvent.sParam, 
			bParam								:= _EmptyEvent.bParam, 
			dParam								:= _EmptyEvent.dParam,
			sFailReason							:= '');
		
		(*Transition*)
		_State									:= 26; // Low Low Alarm - Check abort time
		
	25: (*Low Alarm - Check abort time*)
		_Last_State								:= 25;
		
		(*Action*)
		Warning									:= TRUE;
		Alarm									:= FALSE;
		Abort									:= FALSE;
		
		(*Transition*)
		IF _State_Timer >= AbortTimer THEN
			_State								:= 40; // Abort
		END_IF
		
	26: (*Low Low Alarm - Check abort time*)
		_Last_State								:= 26;
		
		(*Action*)
		Warning									:= TRUE;
		Alarm									:= TRUE;
		Abort									:= FALSE;
		
		(*Transition*)
		IF _State_Timer >= AbortTimer THEN
			_State								:= 41; // Abort
		(*ELSIF PV >= LowLowSP + DB THEN
			_State								:= 21; // Low Low Alarm - Delay
		ELSIF PV >= LowSP + DB THEN
			_State								:= 11; // Low Alarm - Delay*)
		END_IF
		
	40: (*Abort*)
		_Last_State								:= 40;
		
		(*Action*)
		Warning									:= TRUE;
		Alarm									:= FALSE;
		Abort									:= TRUE;
		
		(*Transition*)
		IF PV >= LowSP + DB THEN
			_State								:= 0; // Idle
		END_IF
		
	41: (*Abort*)
		_Last_State								:= 41;
		
		(*Action*)
		Warning									:= TRUE;
		Alarm									:= TRUE;
		Abort									:= TRUE;
		
		(*Transition*)
		IF PV >= LowSP + DB THEN
			_State								:= 0; // Idle
		END_IF
END_CASE

END_FUNCTION_BLOCK

// ---- POUs/3) FB/2) TC/Testing/FB_GUI_TEST_SLTC.TcPOU
FUNCTION_BLOCK FB_GUI_TEST_SLTC
VAR_INPUT
	iLevel :INT;
END_VAR
VAR
	bInitialise : BOOL := FALSE;
	bStartCycle : BOOL := FALSE;
	tCaptureDelay: TIME:= T#1000MS;
	tDelayNextStep: TIME:= T#2000MS;
	tInterval: TIME:= T#200MS;
	
	bCylinderUp : BOOL;
	//iLevel : UINT :=2; 
	
	nState : UINT :=0;
	nCount: INT:=0;
	nNoOfCycle:INT:=1;
	TDelay : TON;
	TDelay1 : TON;
	bUp: BOOL;
	sErr: STRING;
	tempstr : ARRAY[1..4] OF STRING;
	TDelay2 : TON;
	i: INT :=1;
	
	bCylinderOutL1: BOOL;
	bOutL1 : BOOL;
	
	bPBStart : BOOL;
	
	StartPbDly: TON;
	rtStartTrig :F_Trig;
	
	sErrorMsg : STRING;
END_VAR

IF bInitialise THEN
	arrTCLevel[iLevel].stGblParam.bInitialise:=TRUE;
	bInitialise:=FALSE;
END_IF

IF bCylinderUp THEN
	IF (arrTCLevel[iLevel].fbTCLevelSeq.M_nCmptUpDown(bUp, sErr)=10) THEN
		bCylinderUp :=FALSE;
	END_IF
END_IF

IF bMoveShuttle THEN
	sErrorMsg:='';
	bMoveShuttle:=FALSE;
	IF arrTCLevelVIO[iLevel].ipTCCellDoorClosed AND arrTCLevelVIO[iLevel].ipTCCellDoorLock THEN
		IF arrTCLevelVIO[iLevel].ipTCDrawerRetractedinCell THEN
			arrTCLevel[iLevel].stGblParam.bShuttleMoveOut := TRUE;
		ELSE
			arrTCLevel[iLevel].stGblParam.bShuttleMoveIn := TRUE;
		END_IF
	ELSE
		sErrorMsg := 'Door is not lock';
	END_IF
END_IF


(*IF bCylinderOutL1 THEN
	IF (arrTCLevel[iLevel].fbTCLevelSeq.M_nCmptInOut(bOutL1, sErr)=10) THEN
		bCylinderOutL1 :=FALSE;
	END_IF
END_IF*)

(*StartPbDly(in:=(stIO[iLevel].ipStartPB),pt:=T#100MS);
rtStartTrig(Clk:=StartPbDly.Q);
IF rtStartTrig.Q THEN
	bPBStart:=TRUE;
END_IF *)

//bPBStart := stIO[iLevel].ipStartPB;

IF bStartCycle (*OR bPBStart*) THEN //cycle Up down, in out
	CASE nState OF
	 0: 	TDelay(IN:=FALSE);
	 		TDelay1(IN:=FALSE);
			TDelay2(IN:=FALSE);
			i:=1;
			arrTCLevel[iLevel].stGblParam.bShuttleMoveOut := TRUE;
	 		nState := 1;
						
	 1: 	IF arrTCLevel[iLevel].stGblParam.bShuttleMoveOut =FALSE THEN
		 
		 	TDelay1(IN:=TRUE,PT:=tCaptureDelay);
			IF TDelay1.Q THEN
				TDelay2(IN:=TRUE,PT:=tInterval);
				IF TDelay2.Q THEN
										
					TDelay2(IN:=FALSE);
					tempstr[1] := F_concat3('X, ', REAL_TO_STRING(aiXConverted[iLevel]), ', ');
					tempstr[2] := F_concat3('Y, ', REAL_TO_STRING(aiYConverted[iLevel]), ', ');
					tempstr[3] := F_concat3('Z, ', REAL_TO_STRING(aiZConverted[iLevel]), ', ');
					
					tempstr[4] := F_concat3(tempstr[1], tempstr[2], tempstr[3]);
					Logging.fbDebugLog.M_nLogger(1, sSource:='aisensor', F_concat3(INT_TO_STRING(i), ', ', tempstr[4]));
					i := i+1;
				END_IF
				
 
				//END_FOR
			END_IF
			
			
			TDelay(IN:=TRUE,PT:=tDelayNextStep);//after move out, delay before move in
			IF TDelay.Q THEN
				TDelay(IN:=FALSE);
				nState := 2;
			END_IF
			END_IF
			
	 2:		arrTCLevel[iLevel].stGblParam.bShuttleMoveIn := TRUE;
	 		nState := 3;
			
	 3: 	IF arrTCLevel[iLevel].stGblParam.bShuttleMoveIn=FALSE THEN
			TDelay(IN:=TRUE,PT:=tDelayNextStep);//after move out, delay before move in
			IF TDelay.Q THEN
				TDelay(IN:=FALSE);
				nState := 0;
				nCount := nCount +1;
			END_IF	 
	 
			END_IF
	END_CASE
	
	IF nCount> nNoOfCycle(*AND nState =3*) THEN
		bStartCycle := FALSE;
		nCount:=1;
		//bPBStart := FALSE;
		
	END_IF
		
END_IF

END_FUNCTION_BLOCK

// ---- POUs/3) FB/2) TC/Testing/Testing.TcPOU
FUNCTION_BLOCK Testing
VAR_INPUT
END_VAR

VAR_OUTPUT
END_VAR

VAR
	_Input1							: BOOL;
	_Input2							: BOOL;
	_Input3							: BOOL;
	_Input4							: BOOL;
	
	_Result							: INT;
END_VAR

_Result								:= arrTCMultiLevel[1].fbTCMultiLevelSeq.M_GetTIUStatus(
										b0:= _Input1, 
										b1:= _Input2, 
										b2:= _Input3, 
										b3:= _Input4);

END_FUNCTION_BLOCK

// ---- POUs/3) FB/2) TC/Testing/TestManually.TcPOU
 PROGRAM TestManually
VAR
	tTestCmd 				: TON;
	bTIUSlide				: BOOL;
	bSlideOut				: BOOL;
	bDrawer					: BOOL;
	bUpDown					: BOOL;
	bAPAirValve				: BOOL;
	bTesterAirValve			: BOOL;
	bOnOff					: BOOL;
	AP240ACPwr				: BOOL;
	AP240ACPwrPara			: INT;
	bEnableModule			: BOOL;
	bDisableModule			: BOOL;
	bTCCSessionRequest 		: BOOL;
	bTCCSessionStartEnd 	: BOOL;
	bDoorClose				: BOOL;
	bDoorOpen				: BOOL;
	bDPSPower				: BOOL;
	iDPSPowerPara			: INT;
	bLvlAlarmReset			: BOOL;
	bColAlarmReset			: BOOL;
	bCancel					: BOOL;
	bTIUSlideOutRetry		: BOOL;
	bTIUSlideOutCancel		: BOOL;
	bActivateRecipe			: BOOL;
	bValidateRecipe			: BOOL;
	bSetLogFileVerbosity	: BOOL;
	bInitialise				: BOOL;
	bResume					: BOOL;
	
	ClearTCSEvent 		: TON;
	iClearCount   		: INT 		:= 0;
	iTotalClear   		: INT 		:= 20;
	bAutoClearEvent 	: BOOL 		:= FALSE;
	
	iAlarmCodes			: ARRAY[1..NO_OF_LEVEL] OF INT 	:= [1,1,1,1,1,1];
	iAlarmCode			: INT		:= 1;
	iBlinkRate			: INT		:= 1000;
	iSubModule			: INT 		:= 1;
	TestLogName			: STRING	:= '';
	TestCommandID 		: E_TaskName;
	TestModuleID 		: E_ModuleID:=E_ModuleID.NA;
	bTestCommand		: BOOL;	
	TestInteger			: ARRAY[1..10] OF DINT;
	TestString 			: STRING;
	TestBool 			: BOOL;
	iBtnNo				: INT		:= 1;
	i					: INT;
	
	bInitialiseAll 		: BOOL;
	bAlmResetAll 		: BOOL;
	
	tim					: TON;
	miniState			: INT;
	solenoidNumber		: ARRAY [1..10] OF DINT := [1,2,3];
END_VAR

//<HMICommandTest>
	CASE iHMICbCmdSelection OF
		E_Cmd.EnableTester:		 	(*TestBool:=FALSE;*) 	TestInteger[1]:=iAlarmCode; TestString:='';		TestCommandID:=E_TaskName.EnableModule;			TestModuleID:=E_ModuleID.CELL_LA101_TESTER; TestLogName:=CONCAT('EnableModule' ,CONCAT('Level_',INT_TO_STRING(iHMICbLevelSelection)));
		E_Cmd.DisableTester:     	(*TestBool:=FALSE;*) 	TestInteger[1]:=iAlarmCode; TestString:='';		TestCommandID:=E_TaskName.DisableModule;		TestModuleID:=E_ModuleID.CELL_LA101_TESTER; TestLogName:=CONCAT('DisableModule',CONCAT('Level_',INT_TO_STRING(iHMICbLevelSelection)));
	                             
		E_Cmd.EnableTCU:		 	(*TestBool:=FALSE;*) 	TestInteger[1]:=iAlarmCode; TestString:='';		TestCommandID:=E_TaskName.EnableModule;			TestModuleID:=E_ModuleID.CELL_LA101_AP; TestLogName:=CONCAT('EnableTCU' ,CONCAT('Level_',INT_TO_STRING(iHMICbLevelSelection)));
		E_Cmd.DisableTCU:		 	(*TestBool:=FALSE;*) 	TestInteger[1]:=iAlarmCode; TestString:='';		TestCommandID:=E_TaskName.DisableModule;		TestModuleID:=E_ModuleID.CELL_LA101_AP; TestLogName:=CONCAT('DisableTCU',CONCAT('Level_',INT_TO_STRING(iHMICbLevelSelection)));
	                             
		E_Cmd.EnableTII:		 	(*TestBool:=FALSE;*) 	TestInteger[1]:=iAlarmCode; TestString:='';		TestCommandID:=E_TaskName.EnableModule;			TestModuleID:=E_ModuleID.CELL_LA101_TIERII; TestLogName:=CONCAT('EnableTII' ,CONCAT('Level_',INT_TO_STRING(iHMICbLevelSelection)));
		E_Cmd.DisableTII:		 	(*TestBool:=FALSE;*) 	TestInteger[1]:=iAlarmCode; TestString:='';		TestCommandID:=E_TaskName.DisableModule;		TestModuleID:=E_ModuleID.CELL_LA101_TIERII; TestLogName:=CONCAT('DisableTII',CONCAT('Level_',INT_TO_STRING(iHMICbLevelSelection)));

		E_Cmd.INITIALISE:			TestBool:=FALSE; 		TestInteger[1]:=0; TestString:='';				TestCommandID:=E_TaskName.Initialize;				TestModuleID:=LevelModuleID[iHMICbLevelSelection]; 			TestLogName:=CONCAT('Initialize',CONCAT('Level_',INT_TO_STRING(iHMICbLevelSelection)));
		E_Cmd.AlarmReset:		 	(*TestBool:=FALSE;*)	TestInteger[1]:=iAlarmCode; TestString:='';		TestCommandID:=E_TaskName.AlarmReset;				TestModuleID:=LevelModuleID[iHMICbLevelSelection]; 			TestLogName:=CONCAT('AlarmReset',CONCAT('Level_',INT_TO_STRING(iHMICbLevelSelection)));
		E_Cmd.ColumnAlarmReset:	 	(*TestBool:=FALSE;*) 	TestInteger[1]:=iAlarmCode; TestString:='';		TestCommandID:=E_TaskName.AlarmReset;				TestModuleID:=COLUMN_NAME;										 //TestLogName:=CONCAT('Initialize',CONCAT('Level_',INT_TO_STRING(iHMICbLevelSelection)));
		E_Cmd.TIUSlideIn:		 	TestBool:=FALSE; 		TestInteger[1]:=0; TestString:='';				TestCommandID:=E_TaskName.TIUSlideOut;				TestModuleID:=LevelModuleID[iHMICbLevelSelection]; 			TestLogName:=CONCAT('TIUSlideIN',CONCAT('Level_',INT_TO_STRING(iHMICbLevelSelection)));
		E_Cmd.TIUSlideOut:		 	TestBool:=TRUE;			TestInteger[1]:=0; TestString:='';				TestCommandID:=E_TaskName.TIUSlideOut;				TestModuleID:=LevelModuleID[iHMICbLevelSelection]; 			TestLogName:=CONCAT('TIUSlideOut',CONCAT('Level_',INT_TO_STRING(iHMICbLevelSelection)));
		E_Cmd.TIUDrawerUp:		 	TestBool:=TRUE; 		TestInteger[1]:=0; TestString:='';				TestCommandID:=E_TaskName.DrawerUp;					TestModuleID:=LevelModuleID[iHMICbLevelSelection]; 			TestLogName:=CONCAT('DrawerUp',CONCAT('Level_',INT_TO_STRING(iHMICbLevelSelection)));
		E_Cmd.TIUDrawerDown:	 	TestBool:=FALSE; 		TestInteger[1]:=0; TestString:='';            	TestCommandID:=E_TaskName.DrawerUp;					TestModuleID:=LevelModuleID[iHMICbLevelSelection]; 			TestLogName:=CONCAT('DrawerDOWN',CONCAT('Level_',INT_TO_STRING(iHMICbLevelSelection)));
		E_Cmd.TIUSlideOutRetry:  	(*TestBool:=FALSE; 		TestInteger[1]:=0; TestString:='';*)        	TestCommandID:=E_TaskName.TIUSlideOutRetry;			TestModuleID:=LevelModuleID[iHMICbLevelSelection]; 			TestLogName:=CONCAT('TIUSlideOutRetry',CONCAT('Level_',INT_TO_STRING(iHMICbLevelSelection)));
		E_Cmd.TIUSlideOutCancel: 	TestBool:=FALSE; 		TestInteger[1]:=0; TestString:='';            	TestCommandID:=E_TaskName.TIUSlideOutCancel;		TestModuleID:=LevelModuleID[iHMICbLevelSelection]; 			TestLogName:=CONCAT('TIUSlideOutCancel',CONCAT('Level_',INT_TO_STRING(iHMICbLevelSelection)));
		E_Cmd.DPSPowerON:        	TestBool:=FALSE; 		TestInteger[1]:=1; TestString:='';			 	TestCommandID:=E_TaskName.DPSPower;             	TestModuleID:=LevelModuleID[iHMICbLevelSelection]; 			TestLogName:=CONCAT('DPSPowerON',CONCAT('Level_',INT_TO_STRING(iHMICbLevelSelection)));
		E_Cmd.DPSPowerOFF:       	TestBool:=FALSE; 		TestInteger[1]:=0; TestString:='';            	TestCommandID:=E_TaskName.DPSPower;             	TestModuleID:=LevelModuleID[iHMICbLevelSelection]; 			TestLogName:=CONCAT('DPSPowerOFF',CONCAT('Level_',INT_TO_STRING(iHMICbLevelSelection)));
		E_Cmd.DPSPowerAuto:		 	TestBool:=FALSE; 		TestInteger[1]:=2; TestString:='';            	TestCommandID:=E_TaskName.DPSPower;             	TestModuleID:=LevelModuleID[iHMICbLevelSelection]; 			TestLogName:=CONCAT('DPSPowerAUTO',CONCAT('Level_',INT_TO_STRING(iHMICbLevelSelection)));
		E_Cmd.AP240ACPowerON:    	TestBool:=FALSE; 		TestInteger[1]:=1; TestString:='';            	TestCommandID:=E_TaskName.AP240ACPOWER;         	TestModuleID:=LevelModuleID[iHMICbLevelSelection]; 			TestLogName:=CONCAT('AP240ACPwrON',CONCAT('Level_',INT_TO_STRING(iHMICbLevelSelection)));
		E_Cmd.AP240ACPowerOFF:   	TestBool:=FALSE; 		TestInteger[1]:=0; TestString:='';			 	TestCommandID:=E_TaskName.AP240ACPOWER;         	TestModuleID:=LevelModuleID[iHMICbLevelSelection]; 			TestLogName:=CONCAT('AP240ACPwrOFF',CONCAT('Level_',INT_TO_STRING(iHMICbLevelSelection)));
		E_Cmd.APAirValveON:      	TestBool:=TRUE; 		TestInteger[1]:=0; TestString:='';             	TestCommandID:=E_TaskName.APAirValve;           	TestModuleID:=LevelModuleID[iHMICbLevelSelection]; 			TestLogName:=CONCAT('APAirValveON',CONCAT('Level_',INT_TO_STRING(iHMICbLevelSelection)));
		E_Cmd.APAirValveOFF:     	TestBool:=FALSE; 		TestInteger[1]:=0; TestString:='';            	TestCommandID:=E_TaskName.APAirValve;           	TestModuleID:=LevelModuleID[iHMICbLevelSelection]; 			TestLogName:=CONCAT('APAirValveOFF',CONCAT('Level_',INT_TO_STRING(iHMICbLevelSelection)));
		E_Cmd.TstAirValveON:	 	TestBool:=TRUE; 		TestInteger[1]:=0; TestString:='';             	TestCommandID:=E_TaskName.TesterAirValve;       	TestModuleID:=LevelModuleID[iHMICbLevelSelection]; 			TestLogName:=CONCAT('TesterAirValveON',CONCAT('Level_',INT_TO_STRING(iHMICbLevelSelection)));
		E_Cmd.TstAirValveOFF:     	TestBool:=FALSE; 		TestInteger[1]:=0; TestString:='';			 	TestCommandID:=E_TaskName.TesterAirValve;	    	TestModuleID:=LevelModuleID[iHMICbLevelSelection]; 			TestLogName:=CONCAT('TesterAirValveOFF',CONCAT('Level_',INT_TO_STRING(iHMICbLevelSelection)));                 
		E_Cmd.CellDoorOpen:     	TestBool:=FALSE; 		TestInteger[1]:=0; TestString:='';            	TestCommandID:=E_TaskName.DoorOpen;        	 		TestModuleID:=LevelModuleID[iHMICbLevelSelection]; 			TestLogName:=CONCAT('CellDoorOpen',CONCAT('Level_',INT_TO_STRING(iHMICbLevelSelection)));
		E_Cmd.CellDoorClose:	 	TestBool:=TRUE; 		TestInteger[1]:=0; TestString:='';             	TestCommandID:=E_TaskName.DoorClose;       			TestModuleID:=LevelModuleID[iHMICbLevelSelection]; 			TestLogName:=CONCAT('CellDoorClose',CONCAT('Level_',INT_TO_STRING(iHMICbLevelSelection)));
		E_Cmd.CancelBuffer:     	TestBool:=FALSE; 		TestInteger[1]:=0; TestString:='';			 	TestCommandID:=E_TaskName.Cancel;	    			TestModuleID:=E_ModuleID.NA; 								TestLogName:=CONCAT('CancelBuffer',CONCAT('Level_',INT_TO_STRING(iHMICbLevelSelection)));                 
		E_Cmd.TIUSocketAirOn_1:     TestBool:=TRUE; 		TestInteger[1]:=1; TestString:='';             	TestCommandID:=E_TaskName.TIUSocketCoolingAir;		TestModuleID:=LevelModuleID[iHMICbLevelSelection]; 			TestLogName:=CONCAT('TIUSocketCoolingAir_1',CONCAT('Level_',INT_TO_STRING(iHMICbLevelSelection)));
		E_Cmd.TIUSocketAirOn_2:     TestBool:=TRUE; 		TestInteger[1]:=2; TestString:='';             	TestCommandID:=E_TaskName.TIUSocketCoolingAir;		TestModuleID:=LevelModuleID[iHMICbLevelSelection]; 			TestLogName:=CONCAT('TIUSocketCoolingAir_2',CONCAT('Level_',INT_TO_STRING(iHMICbLevelSelection)));
		E_Cmd.TIUSocketAirOff_1:	TestBool:=FALSE; 		TestInteger[1]:=1; TestString:='';             	TestCommandID:=E_TaskName.TIUSocketCoolingAir;		TestModuleID:=LevelModuleID[iHMICbLevelSelection]; 			TestLogName:=CONCAT('TIUSocketCoolingAir_1',CONCAT('Level_',INT_TO_STRING(iHMICbLevelSelection)));
		E_Cmd.TIUSocketAirOff_2:	TestBool:=FALSE; 		TestInteger[1]:=2; TestString:='';             	TestCommandID:=E_TaskName.TIUSocketCoolingAir;		TestModuleID:=LevelModuleID[iHMICbLevelSelection]; 			TestLogName:=CONCAT('TIUSocketCoolingAir_2',CONCAT('Level_',INT_TO_STRING(iHMICbLevelSelection)));		
		E_Cmd.SetLEDON:     		TestBool:=TRUE; 		TestInteger[2]:=0;						TestInteger[1]:=iBtnNo; TestString:='';	TestCommandID:=E_TaskName.SetBlinkRate;	TestModuleID:=LevelModuleID[iHMICbLevelSelection]; TestLogName:=CONCAT(CONCAT('SetLEDON_Btn_0',INT_TO_STRING(iBtnNo)),CONCAT('Level_',INT_TO_STRING(iHMICbLevelSelection)));                 
		E_Cmd.SetLEDOFF:     		TestBool:=FALSE; 		TestInteger[2]:=iBlinkRate; 			TestInteger[1]:=iBtnNo; TestString:='';	TestCommandID:=E_TaskName.SetBlinkRate;	TestModuleID:=LevelModuleID[iHMICbLevelSelection]; TestLogName:=CONCAT(CONCAT('SetLEDON_Btn_0',INT_TO_STRING(iBtnNo)),CONCAT('Level_',INT_TO_STRING(iHMICbLevelSelection)));                 
		E_Cmd.SetLEDBlink:     		TestBool:=TRUE; 		TestInteger[2]:=iBlinkRate; 			TestInteger[1]:=iBtnNo; TestString:='';	TestCommandID:=E_TaskName.SetBlinkRate;	TestModuleID:=LevelModuleID[iHMICbLevelSelection]; TestLogName:=CONCAT(CONCAT('SetLEDBlink_Btn_0',INT_TO_STRING(iBtnNo)),CONCAT('Level_',INT_TO_STRING(iHMICbLevelSelection)));                 
		E_Cmd.DCCellFrontDoorOpen:  TestBool:=FALSE; 		TestInteger[1]:=0; TestString:=''; 				TestCommandID:=E_TaskName.DoorOpen;  				TestModuleID:=LA_FRONT_DOOR_MODULE_ID[iHMICbLevelSelection]; TestLogName:=CONCAT('CellFrontDoorOpen',CONCAT('Level_',INT_TO_STRING(iHMICbLevelSelection)));                
		E_Cmd.DCCellFrontDoorClose: TestBool:=TRUE; 		TestInteger[1]:=0; TestString:='';  			TestCommandID:=E_TaskName.DoorClose; 				TestModuleID:=LA_FRONT_DOOR_MODULE_ID[iHMICbLevelSelection]; TestLogName:=CONCAT('CellFrontDoorClose',CONCAT('Level_',INT_TO_STRING(iHMICbLevelSelection)));     
   		E_Cmd.SetSolenoidValvesON:	TestBool:=TRUE;			TestInteger	:=solenoidNumber; 			TestString:='';				TestCommandID:=E_TaskName.SetSolenoidValves;  		TestModuleID:=LB_LEVEL_MODULE_ID[iHMICbLevelSelection]; 	TestLogName:=CONCAT('SetSolenoidValveON',CONCAT('Level_',INT_TO_STRING(iHMICbLevelSelection)));
		E_Cmd.SetSolenoidValvesOFF:	TestBool:=FALSE;		TestInteger	:=solenoidNumber;			TestString:='';				TestCommandID:=E_TaskName.SetSolenoidValves;  		TestModuleID:=LB_LEVEL_MODULE_ID[iHMICbLevelSelection]; 	TestLogName:=CONCAT('SetSolenoidValveOFF',CONCAT('Level_',INT_TO_STRING(iHMICbLevelSelection)));
		E_Cmd.Secondary24VPowerON:	TestBool:=TRUE; 		TestInteger[1]:=1; TestString:='';            	TestCommandID:=E_TaskName.Secondary24VPower;         	TestModuleID:=LevelModuleID[iHMICbLevelSelection]; 			TestLogName:=CONCAT('Secondary24VPowerON',CONCAT('Level_',INT_TO_STRING(iHMICbLevelSelection)));
		E_Cmd.Secondary24VPowerOFF:	TestBool:=FALSE; 		TestInteger[1]:=0; TestString:='';            	TestCommandID:=E_TaskName.Secondary24VPower;         	TestModuleID:=LevelModuleID[iHMICbLevelSelection]; 			TestLogName:=CONCAT('Secondary24VPowerOFF',CONCAT('Level_',INT_TO_STRING(iHMICbLevelSelection)));

END_CASE                  
//</HMICommandTest>        

//


IF bInitialiseAll THEN
	FOR i:=1 TO NO_OF_LEVEL DO
		arrTACommands.arrTACommands[i].sLogName := CONCAT(CONCAT('Initialise Level[',INT_TO_STRING(i)),']');
		arrTACommands.arrTACommands[i].eTaskName := E_TaskName.Initialize;
		arrTACommands.arrTACommands[i].eModuleID := LevelModuleID[i];
	END_FOR
	arrTCSCommandReady:= FALSE;
	iClearCount := iTotalClear;
	bInitialiseAll := FALSE;
END_IF
	
IF bAlmResetAll THEN
	FOR i:=1 TO NO_OF_LEVEL DO
		arrTACommands.arrTACommands[i].sLogName := CONCAT(CONCAT('Alarm Reset Level[',INT_TO_STRING(i)),']');
		arrTACommands.arrTACommands[i].eTaskName := E_TaskName.AlarmReset;
		arrTACommands.arrTACommands[i].eModuleID := LevelModuleID[i];
		arrTACommands.arrTACommands[1].iParam[1] := iAlarmCodes[i]; //iSubModule;
	END_FOR
	arrTCSCommandReady:= FALSE;
	iClearCount := iTotalClear;
	bAlmResetAll := FALSE;
END_IF
	
//<ManualTest>
	IF bTestCommand   THEN
		arrTACommands.arrTACommands[1].sLogName 	:= TestLogName;
		arrTACommands.arrTACommands[1].eTaskName 	:= TestCommandID;
		arrTACommands.arrTACommands[1].eModuleID 	:= TestModuleID; 
		arrTACommands.arrTACommands[1].iParam[1] 	:= TestInteger[1];
		arrTACommands.arrTACommands[1].iParam[2] 	:= TestInteger[2];
		arrTACommands.arrTACommands[1].iParam		:= TestInteger;
		arrTACommands.arrTACommands[1].sParam[1] 	:= TestString;
		arrTACommands.arrTACommands[1].bParam[1] 	:= TestBool;
		arrTCSCommandReady:= FALSE;
		iClearCount := iTotalClear;
		bTestCommand := FALSE;
	
	ELSIF bInitialise THEN
		arrTACommands.arrTACommands[1].sLogName := 'Initialise_1_TESTER_LA01';
		arrTACommands.arrTACommands[1].eTaskName := E_TaskName.Initialize;
		arrTACommands.arrTACommands[1].eModuleID := TestModuleID;//E_ModuleID.TESTER_LA01;
		//arrTACommands.arrTACommands[1].eModuleID := E_ModuleID.TBOT_R_RFID;
		//arrTACommands.arrTACommands[1].bParam[1] := bSlideOut;
		arrTCSCommandReady:= FALSE;
		iClearCount := iTotalClear;
		bInitialise := FALSE;
	
	ELSIF bActivateRecipe THEN
		arrTACommands.arrTACommands[1].sLogName := 'ActivateRecipe_1_TESTER_LA01';
		arrTACommands.arrTACommands[1].eTaskName := E_TaskName.ActivateRecipe;
		arrTACommands.arrTACommands[1].eModuleID := TestModuleID;//E_ModuleID.TESTER_LA01;
		//arrTACommands.arrTACommands[1].eModuleID := E_ModuleID.TBOT_R_RFID;
		//arrTACommands.arrTACommands[1].bParam[1] := bSlideOut;
		arrTCSCommandReady:= FALSE;
		iClearCount := iTotalClear;
		bActivateRecipe := FALSE;
		
	ELSIF bValidateRecipe THEN
		arrTACommands.arrTACommands[1].sLogName := 'ValidateRecipe_1_TESTER_LA01';
		arrTACommands.arrTACommands[1].eTaskName := E_TaskName.ValidateRecipe;
		arrTACommands.arrTACommands[1].eModuleID := TestModuleID;//E_ModuleID.TESTER_LA01;
		//arrTACommands.arrTACommands[1].eModuleID := E_ModuleID.TBOT_R_RFID;
		arrTACommands.arrTACommands[1].bParam[1] := bSlideOut;
		arrTCSCommandReady:= FALSE;
		iClearCount := iTotalClear;
		bValidateRecipe := FALSE;
	ELSIF bSetLogFileVerbosity THEN
		arrTACommands.arrTACommands[1].sLogName := 'SetLogFileVerbosity_1_TESTER_LA01';
		arrTACommands.arrTACommands[1].eTaskName := E_TaskName.SetLogFileVerbosity;
		arrTACommands.arrTACommands[1].eModuleID := TestModuleID;//E_ModuleID.TESTER_LA01;
		//arrTACommands.arrTACommands[1].eModuleID := E_ModuleID.TBOT_R_RFID;
		//arrTACommands.arrTACommands[1].bParam[1] := bSlideOut;
		arrTCSCommandReady:= FALSE;
		iClearCount := iTotalClear;
		bSetLogFileVerbosity := FALSE;	
	ELSIF bTesterAirValve THEN
		arrTACommands.arrTACommands[1].sLogName := 'TesterAirValve_1_TESTER_LA01';
		arrTACommands.arrTACommands[1].eTaskName := E_TaskName.TesterAirValve;
		arrTACommands.arrTACommands[1].eModuleID := TestModuleID;//E_ModuleID.TESTER_LA01;
		//arrTACommands.arrTACommands[1].eModuleID := E_ModuleID.TBOT_R_RFID;
		arrTACommands.arrTACommands[1].bParam[1] := bOnOff;
		arrTCSCommandReady:= FALSE;
		iClearCount := iTotalClear;
		bTesterAirValve := FALSE;
	ELSIF bAPAirValve THEN
		arrTACommands.arrTACommands[1].sLogName := 'APAirValve_1_TESTER_LA01';
		arrTACommands.arrTACommands[1].eTaskName := E_TaskName.APAirValve;
		arrTACommands.arrTACommands[1].eModuleID := TestModuleID;//E_ModuleID.TESTER_LA01;
		//arrTACommands.arrTACommands[1].eModuleID := E_ModuleID.TBOT_R_RFID;
		arrTACommands.arrTACommands[1].bParam[1] := bOnOff;
		arrTCSCommandReady:= FALSE;
		iClearCount := iTotalClear;
		bAPAirValve := FALSE;
		
	ELSIF bEnableModule THEN
		arrTACommands.arrTACommands[1].sLogName := 'EnableModule_1_TESTER_LA01';
		arrTACommands.arrTACommands[1].eTaskName := E_TaskName.EnableModule;
		arrTACommands.arrTACommands[1].eModuleID := TestModuleID;//E_ModuleID.TESTER_LA01;
		//arrTACommands.arrTACommands[1].eModuleID := E_ModuleID.TBOT_R_RFID;
		//arrTACommands.arrTACommands[1].bParam[1] := bSlideOut;
		arrTCSCommandReady:= FALSE;
		iClearCount := iTotalClear;
		bEnableModule := FALSE;
		
	ELSIF bDisableModule THEN
		arrTACommands.arrTACommands[1].sLogName := 'DisableModule_1_TESTER_LA0';
		arrTACommands.arrTACommands[1].eTaskName := E_TaskName.DisableModule;
		arrTACommands.arrTACommands[1].eModuleID := TestModuleID;//E_ModuleID.TESTER_LA01;
		//arrTACommands.arrTACommands[1].eModuleID := E_ModuleID.TBOT_R_RFID;
		//arrTACommands.arrTACommands[1].bParam[1] := bSlideOut;
		arrTCSCommandReady:= FALSE;
		iClearCount := iTotalClear;
		bDisableModule := FALSE;
	
	ELSIF bTCCSessionRequest THEN
		arrTACommands.arrTACommands[1].sLogName := 'TCCSessionRequest_1_TESTER_LA01';
		arrTACommands.arrTACommands[1].eTaskName := E_TaskName.TCCSessionRequest;
		arrTACommands.arrTACommands[1].eModuleID := TestModuleID;//E_ModuleID.TESTER_LA01;
		arrTACommands.arrTACommands[1].bParam[1] := bTCCSessionStartEnd;
		arrTCSCommandReady:= FALSE;
		iClearCount := iTotalClear;
		bTCCSessionRequest := FALSE;
		
	ELSIF bDPSPower THEN
		arrTACommands.arrTACommands[1].sLogName := 'bDPSPower_1_TESTER_LA01';
		arrTACommands.arrTACommands[1].eTaskName := E_TaskName.DPSPower;
		arrTACommands.arrTACommands[1].eModuleID := TestModuleID;//E_ModuleID.TESTER_LA01;
		//arrTACommands.arrTACommands[1].eModuleID := E_ModuleID.TBOT_R_RFID;
		arrTACommands.arrTACommands[1].iParam[1] := iDPSPowerPara;//(0,1,2)
		arrTCSCommandReady:= FALSE;
		iClearCount := iTotalClear;
		bDPSPower := FALSE;
	ELSIF AP240ACPwr THEN
		arrTACommands.arrTACommands[1].sLogName := 'AP240ACPower_1_TESTER_LA01';
		arrTACommands.arrTACommands[1].eTaskName := E_TaskName.AP240ACPOWER;
		arrTACommands.arrTACommands[1].eModuleID := TestModuleID;//E_ModuleID.TESTER_LA01;
		//arrTACommands.arrTACommands[1].eModuleID := E_ModuleID.TBOT_R_RFID;
		arrTACommands.arrTACommands[1].iParam[1] := AP240ACPwrPara;//(0,1,2)
		arrTCSCommandReady:= FALSE;
		iClearCount := iTotalClear;
		AP240ACPwr := FALSE;
		
	ELSIF bDoorClose THEN
		arrTACommands.arrTACommands[1].sLogName := 'DoorCloseRequest_1_TESTER_LA01';
		arrTACommands.arrTACommands[1].eTaskName := E_TaskName.DoorClose;
		arrTACommands.arrTACommands[1].eModuleID := TestModuleID;//E_ModuleID.TESTER_LA01;
		//arrTACommands.arrTACommands[1].eModuleID := E_ModuleID.TBOT_R_RFID;
		//arrTACommands.arrTACommands[1].bParam[1] := bSlideOut;
		arrTCSCommandReady:= FALSE;
		iClearCount := iTotalClear;
		bDoorClose := FALSE;
		
	ELSIF bDoorOpen THEN
		arrTACommands.arrTACommands[1].sLogName := 'DoorOpenRequest_1_TESTER_LA01';
		arrTACommands.arrTACommands[1].eTaskName := E_TaskName.DoorOpen;
		arrTACommands.arrTACommands[1].eModuleID := TestModuleID;//E_ModuleID.TESTER_LA01;
		//arrTACommands.arrTACommands[1].eModuleID := E_ModuleID.TBOT_R_RFID;
		//arrTACommands.arrTACommands[1].bParam[1] := bSlideOut;
		arrTCSCommandReady:= FALSE;
		iClearCount := iTotalClear;
		bDoorOpen := FALSE;
	ELSIF bDrawer THEN
		arrTACommands.arrTACommands[1].sLogName := 'DrawerUp_1_TESTER_LA01';
		arrTACommands.arrTACommands[1].eTaskName := E_TaskName.DrawerUp;
		arrTACommands.arrTACommands[1].eModuleID := TestModuleID;//E_ModuleID.TESTER_LA01;
		//arrTACommands.arrTACommands[1].eModuleID := E_ModuleID.TBOT_R_RFID;
		arrTACommands.arrTACommands[1].bParam[1] := bUpDown;
		arrTCSCommandReady:= FALSE;
		iClearCount := iTotalClear;
		bDrawer := FALSE;	
	ELSIF bTIUSlide THEN
		arrTACommands.arrTACommands[1].sLogName := 'TIUSlideOut_1_TESTER_LA01';
		arrTACommands.arrTACommands[1].eTaskName := E_TaskName.TIUSlideOut;
		arrTACommands.arrTACommands[1].eModuleID := TestModuleID;//E_ModuleID.TESTER_LA01;
		//arrTACommands.arrTACommands[1].eModuleID := E_ModuleID.TBOT_R_RFID;
		arrTACommands.arrTACommands[1].bParam[1] := bSlideOut;
		arrTCSCommandReady:= FALSE;
		iClearCount := iTotalClear;
		bTIUSlide := FALSE;
	ELSIF bTIUSlideOutRetry THEN
		arrTACommands.arrTACommands[1].sLogName := 'TIUSlideOutRetry_1_TESTER_LA01';
		arrTACommands.arrTACommands[1].eTaskName := E_TaskName.TIUSlideOutRetry;
		arrTACommands.arrTACommands[1].eModuleID := TestModuleID;//E_ModuleID.TESTER_LA01;
		arrTACommands.arrTACommands[1].bParam[1] := bSlideOut;
		arrTCSCommandReady:= FALSE;
		iClearCount := iTotalClear;
		bTIUSlideOutRetry := FALSE;
	ELSIF bTIUSlideOutCancel THEN
		arrTACommands.arrTACommands[1].sLogName := 'TIUSlideOutCancel_1_TESTER_LA01';
		arrTACommands.arrTACommands[1].eTaskName := E_TaskName.TIUSlideOutCancel;
		arrTACommands.arrTACommands[1].eModuleID := TestModuleID;//E_ModuleID.TESTER_LA01;
		//arrTACommands.arrTACommands[1].bParam[1] := bSlideOut;
		arrTCSCommandReady:= FALSE;
		iClearCount := iTotalClear;
		bTIUSlideOutCancel := FALSE;
		
	ELSIF bCancel THEN
		arrTACommands.arrTACommands[1].sLogName := 'Cancel_NA [Buffer Clear]';
		arrTACommands.arrTACommands[1].eTaskName := E_TaskName.Cancel;
		arrTACommands.arrTACommands[1].eModuleID := E_ModuleID.NA;
		arrTACommands.arrTACommands[1].bParam[1] := 1;
		arrTCSCommandReady:= FALSE;
		iClearCount := iTotalClear;
		bCancel := FALSE;
	
	ELSIF bLvlAlarmReset THEN
		arrTACommands.arrTACommands[1].sLogName := 'LevelAlarmReset';
		arrTACommands.arrTACommands[1].eTaskName := E_TaskName.AlarmReset;
		arrTACommands.arrTACommands[1].eModuleID := TestModuleID;//E_ModuleID.TESTER_LA01;
		arrTACommands.arrTACommands[1].iParam[1] := iAlarmCode; //iSubModule;
		//arrTACommands.arrTACommands[1].iParam[2] := iAlarmCode;
		//arrTACommands.arrTACommands[1].iParam := F_ArrayInt(iParam:= arrTACommands.arrTACommands[1].iParam, iParam1 := iAlarmCode);
		arrTCSCommandReady:= FALSE;
		iClearCount := iTotalClear;
		bLvlAlarmReset := FALSE;
		
	ELSIF bColAlarmReset THEN
		arrTACommands.arrTACommands[1].sLogName := TestLogName;
		arrTACommands.arrTACommands[1].eTaskName := TestCommandID;
		arrTACommands.arrTACommands[1].eModuleID := COLUMN_NAME;
		arrTACommands.arrTACommands[1].iParam[1] := iAlarmCode; //iSubModule;
		//arrTACommands.arrTACommands[1].iParam[2] := iAlarmCode;
		//arrTACommands.arrTACommands[1].iParam := F_ArrayInt(iParam:= arrTACommands.arrTACommands[1].iParam, iParam1 := iAlarmCode);
		arrTCSCommandReady:= FALSE;
		iClearCount := iTotalClear;
		bColAlarmReset := FALSE;
	
	ELSIF bResume THEN
		arrTACommands.arrTACommands[1].sLogName := 'Resume_1_TESTER_LA01';
		arrTACommands.arrTACommands[1].eTaskName := E_TaskName.Resume;
		arrTACommands.arrTACommands[1].eModuleID := TestModuleID;//E_ModuleID.TESTER_LA01;
		//arrTACommands.arrTACommands[1].bParam[1] := bSlideOut;
		arrTCSCommandReady:= FALSE;
		iClearCount := iTotalClear;
		bResume := FALSE;
	(**)	
	END_IF
//</ManualTest>	




IF bAutoClearEvent THEN
	iClearCount := iTotalClear;
END_IF

//Ensure the arrTCSEventTriggered[] are fully cleared
ClearTCSEvent(IN:=(iClearCount > 0), PT:=T#100MS);
IF ClearTCSEvent.Q THEN
	ClearTCSEvent(IN:=FALSE);
	iClearCount := iClearCount - 1;
	arrTCSEventTriggered:= FALSE;
	
END_IF
	
tTestCmd(IN:=FALSE, PT:=T#5S);
IF tTestCmd.Q THEN
	tTestCmd(IN:=FALSE);
	bTIUSlide :=TRUE;
END_IF

METHOD TestCommand : Bool
VAR_INPUT
	sLogName:STRING;
	eTaskName:E_TaskName;
	eModuleID:E_ModuleID;
END_VAR
END_METHOD

END_PROGRAM

